(* Logix 5000 project; controller TBEN_Lx_8IOL_AOI_V0_2 vendor 1 type 14 code 176 rev 32.11; software revision 32.00; part 6 of 11 *)

           TBEN_L4_8IOL:C.Data[144].6   // IO-Link Port 8 - Device ID (INT bit22)
           TBEN_L4_8IOL:C.Data[144].7   // IO-Link Port 8 - Device ID (INT bit23)
           TBEN_L4_8IOL:C.Data[145]   // IO-Link Port 8 - Device ID
           TBEN_L4_8IOL:C.Data[145].0   // IO-Link Port 8 - Device ID (INT bit24)
           TBEN_L4_8IOL:C.Data[145].1   // IO-Link Port 8 - Device ID (INT bit25)
           TBEN_L4_8IOL:C.Data[145].2   // IO-Link Port 8 - Device ID (INT bit26)
           TBEN_L4_8IOL:C.Data[145].3   // IO-Link Port 8 - Device ID (INT bit27)
           TBEN_L4_8IOL:C.Data[145].4   // IO-Link Port 8 - Device ID (INT bit28)
           TBEN_L4_8IOL:C.Data[145].5   // IO-Link Port 8 - Device ID (INT bit29)
           TBEN_L4_8IOL:C.Data[145].6   // IO-Link Port 8 - Device ID (INT bit30)
           TBEN_L4_8IOL:C.Data[145].7   // IO-Link Port 8 - Device ID (INT bit31)
           TBEN_L4_8IOL:C.Data[146]   // VAUX1 Pin1 C0 (Ch0/1)
           TBEN_L4_8IOL:C.Data[146].0   // VAUX1 Pin1 C0 (Ch0/1) (ENUM bit0): 00=24 VDC, 01=switchable
           TBEN_L4_8IOL:C.Data[146].1   // VAUX1 Pin1 C0 (Ch0/1) (ENUM bit1): 10=off
           TBEN_L4_8IOL:C.Data[146].2   // Reserved
           TBEN_L4_8IOL:C.Data[146].3   // Reserved
           TBEN_L4_8IOL:C.Data[146].4   // Reserved
           TBEN_L4_8IOL:C.Data[146].5   // Reserved
           TBEN_L4_8IOL:C.Data[146].6   // Reserved
           TBEN_L4_8IOL:C.Data[146].7   // Reserved
           TBEN_L4_8IOL:C.Data[147]   // VAUX1 Pin1 C1 (Ch2/3)
           TBEN_L4_8IOL:C.Data[147].0   // VAUX1 Pin1 C1 (Ch2/3) (ENUM bit0): 00=24 VDC, 01=switchable
           TBEN_L4_8IOL:C.Data[147].1   // VAUX1 Pin1 C1 (Ch2/3) (ENUM bit1): 10=off
           TBEN_L4_8IOL:C.Data[147].2   // Reserved
           TBEN_L4_8IOL:C.Data[147].3   // Reserved
           TBEN_L4_8IOL:C.Data[147].4   // Reserved
           TBEN_L4_8IOL:C.Data[147].5   // Reserved
           TBEN_L4_8IOL:C.Data[147].6   // Reserved
           TBEN_L4_8IOL:C.Data[147].7   // Reserved
           TBEN_L4_8IOL:C.Data[148]   // VAUX1 Pin1 C2 (Ch4/5)
           TBEN_L4_8IOL:C.Data[148].0   // VAUX1 Pin1 C2 (Ch4/5) (ENUM bit0): 00=24 VDC, 01=switchable
           TBEN_L4_8IOL:C.Data[148].1   // VAUX1 Pin1 C2 (Ch4/5) (ENUM bit1): 10=off
           TBEN_L4_8IOL:C.Data[148].2   // Reserved
           TBEN_L4_8IOL:C.Data[148].3   // Reserved
           TBEN_L4_8IOL:C.Data[148].4   // Reserved
           TBEN_L4_8IOL:C.Data[148].5   // Reserved
           TBEN_L4_8IOL:C.Data[148].6   // Reserved
           TBEN_L4_8IOL:C.Data[148].7   // Reserved
           TBEN_L4_8IOL:C.Data[149]   // VAUX1 Pin1 C3 (Ch6/7)
           TBEN_L4_8IOL:C.Data[149].0   // VAUX1 Pin1 C3 (Ch6/7) (ENUM bit0): 00=24 VDC, 01=switchable
           TBEN_L4_8IOL:C.Data[149].1   // VAUX1 Pin1 C3 (Ch6/7) (ENUM bit1): 10=off
           TBEN_L4_8IOL:C.Data[149].2   // Reserved
           TBEN_L4_8IOL:C.Data[149].3   // Reserved
           TBEN_L4_8IOL:C.Data[149].4   // Reserved
           TBEN_L4_8IOL:C.Data[149].5   // Reserved
           TBEN_L4_8IOL:C.Data[149].6   // Reserved
           TBEN_L4_8IOL:C.Data[149].7   // Reserved
           TBEN_L4_8IOL:C.Data[14]   // DXP 1 - Activate output
           TBEN_L4_8IOL:C.Data[14].0   // DXP 1 - Activate output (ENUM bit0): 0=no, 1=yes
           TBEN_L4_8IOL:C.Data[14].1   // Reserved
           TBEN_L4_8IOL:C.Data[14].2   // Reserved
           TBEN_L4_8IOL:C.Data[14].3   // Reserved
           TBEN_L4_8IOL:C.Data[14].4   // Reserved
           TBEN_L4_8IOL:C.Data[14].5   // Reserved
           TBEN_L4_8IOL:C.Data[14].6   // Reserved
           TBEN_L4_8IOL:C.Data[14].7   // Reserved
           TBEN_L4_8IOL:C.Data[150]   // VAUX1 Pin1 C4 (Ch8)
           TBEN_L4_8IOL:C.Data[150].0   // VAUX1 Pin1 C4 (Ch8) (ENUM bit0): 00=24 VDC, 01=switchable
           TBEN_L4_8IOL:C.Data[150].1   // VAUX1 Pin1 C4 (Ch8) (ENUM bit1): 10=off
           TBEN_L4_8IOL:C.Data[150].2   // Reserved
           TBEN_L4_8IOL:C.Data[150].3   // Reserved
           TBEN_L4_8IOL:C.Data[150].4   // Reserved
           TBEN_L4_8IOL:C.Data[150].5   // Reserved
           TBEN_L4_8IOL:C.Data[150].6   // Reserved
           TBEN_L4_8IOL:C.Data[150].7   // Reserved
           TBEN_L4_8IOL:C.Data[151]   // VAUX2 Pin2 C4 (Ch9)
           TBEN_L4_8IOL:C.Data[151].0   // VAUX2 Pin2 C4 (Ch9) (ENUM bit0): 00=24 VDC, 01=switchable
           TBEN_L4_8IOL:C.Data[151].1   // VAUX2 Pin2 C4 (Ch9) (ENUM bit1): 10=off
           TBEN_L4_8IOL:C.Data[151].2   // Reserved
           TBEN_L4_8IOL:C.Data[151].3   // Reserved
           TBEN_L4_8IOL:C.Data[151].4   // Reserved
           TBEN_L4_8IOL:C.Data[151].5   // Reserved
           TBEN_L4_8IOL:C.Data[151].6   // Reserved
           TBEN_L4_8IOL:C.Data[151].7   // Reserved
           TBEN_L4_8IOL:C.Data[152]   // VAUX1 Pin1 C5 (Ch10)
           TBEN_L4_8IOL:C.Data[152].0   // VAUX1 Pin1 C5 (Ch10) (ENUM bit0): 00=24 VDC, 01=switchable
           TBEN_L4_8IOL:C.Data[152].1   // VAUX1 Pin1 C5 (Ch10) (ENUM bit1): 10=off
           TBEN_L4_8IOL:C.Data[152].2   // Reserved
           TBEN_L4_8IOL:C.Data[152].3   // Reserved
           TBEN_L4_8IOL:C.Data[152].4   // Reserved
           TBEN_L4_8IOL:C.Data[152].5   // Reserved
           TBEN_L4_8IOL:C.Data[152].6   // Reserved
           TBEN_L4_8IOL:C.Data[152].7   // Reserved
           TBEN_L4_8IOL:C.Data[153]   // VAUX2 Pin2 C5 (Ch11)
           TBEN_L4_8IOL:C.Data[153].0   // VAUX2 Pin2 C5 (Ch11) (ENUM bit0): 00=24 VDC, 01=switchable
           TBEN_L4_8IOL:C.Data[153].1   // VAUX2 Pin2 C5 (Ch11) (ENUM bit1): 10=off
           TBEN_L4_8IOL:C.Data[153].2   // Reserved
           TBEN_L4_8IOL:C.Data[153].3   // Reserved
           TBEN_L4_8IOL:C.Data[153].4   // Reserved
           TBEN_L4_8IOL:C.Data[153].5   // Reserved
           TBEN_L4_8IOL:C.Data[153].6   // Reserved
           TBEN_L4_8IOL:C.Data[153].7   // Reserved
           TBEN_L4_8IOL:C.Data[154]   // VAUX1 Pin1 C6 (Ch12)
           TBEN_L4_8IOL:C.Data[154].0   // VAUX1 Pin1 C6 (Ch12) (ENUM bit0): 00=24 VDC, 01=switchable
           TBEN_L4_8IOL:C.Data[154].1   // VAUX1 Pin1 C6 (Ch12) (ENUM bit1): 10=off
           TBEN_L4_8IOL:C.Data[154].2   // Reserved
           TBEN_L4_8IOL:C.Data[154].3   // Reserved
           TBEN_L4_8IOL:C.Data[154].4   // Reserved
           TBEN_L4_8IOL:C.Data[154].5   // Reserved
           TBEN_L4_8IOL:C.Data[154].6   // Reserved
           TBEN_L4_8IOL:C.Data[154].7   // Reserved
           TBEN_L4_8IOL:C.Data[155]   // VAUX2 Pin2 C6 (Ch13)
           TBEN_L4_8IOL:C.Data[155].0   // VAUX2 Pin2 C6 (Ch13) (ENUM bit0): 00=24 VDC, 01=switchable
           TBEN_L4_8IOL:C.Data[155].1   // VAUX2 Pin2 C6 (Ch13) (ENUM bit1): 10=off
           TBEN_L4_8IOL:C.Data[155].2   // Reserved
           TBEN_L4_8IOL:C.Data[155].3   // Reserved
           TBEN_L4_8IOL:C.Data[155].4   // Reserved
           TBEN_L4_8IOL:C.Data[155].5   // Reserved
           TBEN_L4_8IOL:C.Data[155].6   // Reserved
           TBEN_L4_8IOL:C.Data[155].7   // Reserved
           TBEN_L4_8IOL:C.Data[156]   // VAUX1 Pin1 C7 (Ch14)
           TBEN_L4_8IOL:C.Data[156].0   // VAUX1 Pin1 C7 (Ch14) (ENUM bit0): 00=24 VDC, 01=switchable
           TBEN_L4_8IOL:C.Data[156].1   // VAUX1 Pin1 C7 (Ch14) (ENUM bit1): 10=off
           TBEN_L4_8IOL:C.Data[156].2   // Reserved
           TBEN_L4_8IOL:C.Data[156].3   // Reserved
           TBEN_L4_8IOL:C.Data[156].4   // Reserved
           TBEN_L4_8IOL:C.Data[156].5   // Reserved
           TBEN_L4_8IOL:C.Data[156].6   // Reserved
           TBEN_L4_8IOL:C.Data[156].7   // Reserved
           TBEN_L4_8IOL:C.Data[157]   // VAUX2 Pin2 C7 (Ch15)
           TBEN_L4_8IOL:C.Data[157].0   // VAUX2 Pin2 C7 (Ch15) (ENUM bit0): 00=24 VDC, 01=switchable
           TBEN_L4_8IOL:C.Data[157].1   // VAUX2 Pin2 C7 (Ch15) (ENUM bit1): 10=off
           TBEN_L4_8IOL:C.Data[157].2   // Reserved
           TBEN_L4_8IOL:C.Data[157].3   // Reserved
           TBEN_L4_8IOL:C.Data[157].4   // Reserved
           TBEN_L4_8IOL:C.Data[157].5   // Reserved
           TBEN_L4_8IOL:C.Data[157].6   // Reserved
           TBEN_L4_8IOL:C.Data[157].7   // Reserved
           TBEN_L4_8IOL:C.Data[15]   // DXP 3 - Activate output
           TBEN_L4_8IOL:C.Data[15].0   // DXP 3 - Activate output (ENUM bit0): 0=no, 1=yes
           TBEN_L4_8IOL:C.Data[15].1   // Reserved
           TBEN_L4_8IOL:C.Data[15].2   // Reserved
           TBEN_L4_8IOL:C.Data[15].3   // Reserved
           TBEN_L4_8IOL:C.Data[15].4   // Reserved
           TBEN_L4_8IOL:C.Data[15].5   // Reserved
           TBEN_L4_8IOL:C.Data[15].6   // Reserved
           TBEN_L4_8IOL:C.Data[15].7   // Reserved
           TBEN_L4_8IOL:C.Data[16]   // DXP 5 - Activate output
           TBEN_L4_8IOL:C.Data[16].0   // DXP 5 - Activate output (ENUM bit0): 0=no, 1=yes
           TBEN_L4_8IOL:C.Data[16].1   // Reserved
           TBEN_L4_8IOL:C.Data[16].2   // Reserved
           TBEN_L4_8IOL:C.Data[16].3   // Reserved
           TBEN_L4_8IOL:C.Data[16].4   // Reserved
           TBEN_L4_8IOL:C.Data[16].5   // Reserved
           TBEN_L4_8IOL:C.Data[16].6   // Reserved
           TBEN_L4_8IOL:C.Data[16].7   // Reserved
           TBEN_L4_8IOL:C.Data[17]   // DXP 7 - Activate output
           TBEN_L4_8IOL:C.Data[17].0   // DXP 7 - Activate output (ENUM bit0): 0=no, 1=yes
           TBEN_L4_8IOL:C.Data[17].1   // Reserved
           TBEN_L4_8IOL:C.Data[17].2   // Reserved
           TBEN_L4_8IOL:C.Data[17].3   // Reserved
           TBEN_L4_8IOL:C.Data[17].4   // Reserved
           TBEN_L4_8IOL:C.Data[17].5   // Reserved
           TBEN_L4_8IOL:C.Data[17].6   // Reserved
           TBEN_L4_8IOL:C.Data[17].7   // Reserved
           TBEN_L4_8IOL:C.Data[18]   // IO-Link Port 1 - Operation mode
           TBEN_L4_8IOL:C.Data[18].0   // IO-Link Port 1 - Operation mode (ENUM bit0): 0000=IO-Link without validation, 0001=IO-Link with family compatible device
           TBEN_L4_8IOL:C.Data[18].1   // IO-Link Port 1 - Operation mode (ENUM bit1): 0010=IO-Link with compatible device, 0011=IO-Link with identical device
           TBEN_L4_8IOL:C.Data[18].2   // IO-Link Port 1 - Operation mode (ENUM bit2): 0100=DI (with parameter access)
           TBEN_L4_8IOL:C.Data[18].3   // IO-Link Port 1 - Operation mode (ENUM bit3): 1000=DI
           TBEN_L4_8IOL:C.Data[18].4   // Reserved
           TBEN_L4_8IOL:C.Data[18].5   // Reserved
           TBEN_L4_8IOL:C.Data[18].6   // Reserved
           TBEN_L4_8IOL:C.Data[18].7   // Reserved
           TBEN_L4_8IOL:C.Data[19]   // IO-Link Port 1 - Data storage mode
           TBEN_L4_8IOL:C.Data[19].0   // IO-Link Port 1 - Data storage mode (ENUM bit0): 00=activated, 01=overwrite
           TBEN_L4_8IOL:C.Data[19].1   // IO-Link Port 1 - Data storage mode (ENUM bit1): 10=read in, 11=deactivated, clear
           TBEN_L4_8IOL:C.Data[19].2   // Reserved
           TBEN_L4_8IOL:C.Data[19].3   // Reserved
           TBEN_L4_8IOL:C.Data[19].4   // Reserved
           TBEN_L4_8IOL:C.Data[19].5   // Reserved
           TBEN_L4_8IOL:C.Data[19].6   // Reserved
           TBEN_L4_8IOL:C.Data[19].7   // Reserved
           TBEN_L4_8IOL:C.Data[1]   // Reserved
           TBEN_L4_8IOL:C.Data[20]   // IO-Link Port 1 - Cycle time
           TBEN_L4_8IOL:C.Data[20].0   // IO-Link Port 1 - Cycle time (ENUM bit0): 00000000=automatic, 00010000=1.6 ms, 00011000=2.4 ms, 00100000=3.2 ms, 00101000=4.0 ms, 00110000=4.8 ms, 00111000=5.6 ms, 01000000=6.4 ms, 01000010=7.2 ms, 01000100=8.0 ms, 01000110=8.8 ms, 01001000=9.6 ms
           TBEN_L4_8IOL:C.Data[20].1   // IO-Link Port 1 - Cycle time (ENUM bit1): 01001010=10.4 ms, 01001100=11.2 ms, 01001110=12.0 ms, 01010000=12.8 ms, 01010100=14.4 ms, 01011000=16.0 ms, 01011100=17.6 ms, 01100000=19.2 ms, 01100100=20.8 ms, 01101000=22.4 ms, 01101100=24.0 ms, 01110000=25.6 ms
           TBEN_L4_8IOL:C.Data[20].2   // IO-Link Port 1 - Cycle time (ENUM bit2): 01110100=27.2 ms, 01111000=28.8 ms, 01111100=30.4 ms, 10000000=32.0 ms, 10000001=33.6 ms, 10000010=35.2 ms, 10000011=36.8 ms, 10000100=38.4 ms, 10000101=40.0 ms, 10000110=41.6 ms, 10000111=43.2 ms, 10001000=44.8 ms
           TBEN_L4_8IOL:C.Data[20].3   // IO-Link Port 1 - Cycle time (ENUM bit3): 10001001=46.4 ms, 10001010=48.0 ms, 10001011=49.6 ms, 10001100=51.2 ms, 10001101=52.8 ms, 10001110=54.4 ms, 10001111=56.0 ms, 10010000=57.6 ms, 10010001=59.2 ms, 10010010=60.8 ms, 10010011=62.4 ms, 10010100=64.0 ms
           TBEN_L4_8IOL:C.Data[20].4   // IO-Link Port 1 - Cycle time (ENUM bit4): 10010101=65.6 ms, 10010110=67.2 ms, 10010111=68.8 ms, 10011000=70.4 ms, 10011001=72.0 ms, 10011010=73.6 ms, 10011011=75.2 ms, 10011100=76.8 ms, 10011101=78.4 ms, 10011110=80.0 ms, 10011111=81.6 ms
           TBEN_L4_8IOL:C.Data[20].5   // IO-Link Port 1 - Cycle time (ENUM bit5): 10100000=83.2 ms, 10100001=84.8 ms, 10100010=86.4 ms, 10100011=88.0 ms, 10100100=89.6 ms, 10100101=91.2 ms, 10100110=92.8 ms, 10100111=94.4 ms, 10101000=96.0 ms, 10101001=97.6 ms, 10101010=99.2 ms
           TBEN_L4_8IOL:C.Data[20].6   // IO-Link Port 1 - Cycle time (ENUM bit6): 10101011=100.8 ms, 10101100=102.4 ms, 10101101=104.0 ms, 10101110=105.6 ms, 10101111=107.2 ms, 10110000=108.8 ms, 10110001=110.4 ms, 10110010=112.0 ms, 10110011=113.6 ms, 10110100=115.2 ms, 10110101=116.8 ms
           TBEN_L4_8IOL:C.Data[20].7   // IO-Link Port 1 - Cycle time (ENUM bit7): 10110110=118.4 ms, 10110111=120.0 ms, 10111000=121.6 ms, 10111001=123.2 ms, 10111010=124.8 ms, 10111011=126.4 ms, 10111100=128.0 ms, 10111101=129.6 ms, 10111110=131.2 ms, 10111111=132.8 ms, 11111111=automatic, compatible
           TBEN_L4_8IOL:C.Data[21]   // IO-Link Port 1 - Revision
           TBEN_L4_8IOL:C.Data[21].0   // IO-Link Port 1 - Revision (ENUM bit0): 0=automatic, 1=V1.0
           TBEN_L4_8IOL:C.Data[21].1   // Reserved
           TBEN_L4_8IOL:C.Data[21].2   // Reserved
           TBEN_L4_8IOL:C.Data[21].3   // Reserved
           TBEN_L4_8IOL:C.Data[21].4   // Reserved
           TBEN_L4_8IOL:C.Data[21].5   // Reserved
           TBEN_L4_8IOL:C.Data[21].6   // Reserved
           TBEN_L4_8IOL:C.Data[21].7   // Reserved
           TBEN_L4_8IOL:C.Data[22]   // IO-Link Port 1 - Activate Quick Start-Up
           TBEN_L4_8IOL:C.Data[22].0   // IO-Link Port 1 - Activate Quick Start-Up (ENUM bit0): 0=no, 1=yes
           TBEN_L4_8IOL:C.Data[22].1   // Reserved
           TBEN_L4_8IOL:C.Data[22].2   // Reserved
           TBEN_L4_8IOL:C.Data[22].3   // Reserved
           TBEN_L4_8IOL:C.Data[22].4   // Reserved
           TBEN_L4_8IOL:C.Data[22].5   // Reserved
           TBEN_L4_8IOL:C.Data[22].6   // Reserved
           TBEN_L4_8IOL:C.Data[22].7   // Reserved
           TBEN_L4_8IOL:C.Data[23]   // IO-Link Port 1 - Device parametrization via GSD
           TBEN_L4_8IOL:C.Data[23].0   // IO-Link Port 1 - Device parametrization via GSD (ENUM bit0): 0=inactive, 1=active
           TBEN_L4_8IOL:C.Data[23].1   // Reserved
           TBEN_L4_8IOL:C.Data[23].2   // Reserved
           TBEN_L4_8IOL:C.Data[23].3   // Reserved
           TBEN_L4_8IOL:C.Data[23].4   // Reserved
           TBEN_L4_8IOL:C.Data[23].5   // Reserved
           TBEN_L4_8IOL:C.Data[23].6   // Reserved
           TBEN_L4_8IOL:C.Data[23].7   // Reserved
           TBEN_L4_8IOL:C.Data[24]   // IO-Link Port 1 - Process input data invalid
           TBEN_L4_8IOL:C.Data[24].0   // IO-Link Port 1 - Process input data invalid (ENUM bit0): 0=diagnostic generated, 1=no diagnostic generated
           TBEN_L4_8IOL:C.Data[24].1   // Reserved
           TBEN_L4_8IOL:C.Data[24].2   // Reserved
           TBEN_L4_8IOL:C.Data[24].3   // Reserved
           TBEN_L4_8IOL:C.Data[24].4   // Reserved
           TBEN_L4_8IOL:C.Data[24].5   // Reserved
           TBEN_L4_8IOL:C.Data[24].6   // Reserved
           TBEN_L4_8IOL:C.Data[24].7   // Reserved
           TBEN_L4_8IOL:C.Data[25]   // IO-Link Port 1 - Deactivate diagnostics
           TBEN_L4_8IOL:C.Data[25].0   // IO-Link Port 1 - Deactivate diagnostics (ENUM bit0): 00=no, 01=notifications
           TBEN_L4_8IOL:C.Data[25].1   // IO-Link Port 1 - Deactivate diagnostics (ENUM bit1): 10=notifications and warnings, 11=yes
           TBEN_L4_8IOL:C.Data[25].2   // Reserved
           TBEN_L4_8IOL:C.Data[25].3   // Reserved
           TBEN_L4_8IOL:C.Data[25].4   // Reserved
           TBEN_L4_8IOL:C.Data[25].5   // Reserved
           TBEN_L4_8IOL:C.Data[25].6   // Reserved
           TBEN_L4_8IOL:C.Data[25].7   // Reserved
           TBEN_L4_8IOL:C.Data[26]   // IO-Link Port 1 - Input data mapping
           TBEN_L4_8IOL:C.Data[26].0   // IO-Link Port 1 - Input data mapping (ENUM bit0): 00=direct, 01=swap 16 bit
           TBEN_L4_8IOL:C.Data[26].1   // IO-Link Port 1 - Input data mapping (ENUM bit1): 10=swap 32 bit, 11=swap
           TBEN_L4_8IOL:C.Data[26].2   // Reserved
           TBEN_L4_8IOL:C.Data[26].3   // Reserved
           TBEN_L4_8IOL:C.Data[26].4   // Reserved
           TBEN_L4_8IOL:C.Data[26].5   // Reserved
           TBEN_L4_8IOL:C.Data[26].6   // Reserved
           TBEN_L4_8IOL:C.Data[26].7   // Reserved
           TBEN_L4_8IOL:C.Data[27]   // IO-Link Port 1 - Output data mapping
           TBEN_L4_8IOL:C.Data[27].0   // IO-Link Port 1 - Output data mapping (ENUM bit0): 00=direct, 01=swap 16 bit
           TBEN_L4_8IOL:C.Data[27].1   // IO-Link Port 1 - Output data mapping (ENUM bit1): 10=swap 32 bit, 11=swap
           TBEN_L4_8IOL:C.Data[27].2   // Reserved
           TBEN_L4_8IOL:C.Data[27].3   // Reserved
           TBEN_L4_8IOL:C.Data[27].4   // Reserved
           TBEN_L4_8IOL:C.Data[27].5   // Reserved
           TBEN_L4_8IOL:C.Data[27].6   // Reserved
           TBEN_L4_8IOL:C.Data[27].7   // Reserved
           TBEN_L4_8IOL:C.Data[28]   // IO-Link Port 1 - Vendor ID
           TBEN_L4_8IOL:C.Data[28].0   // IO-Link Port 1 - Vendor ID (INT bit0)
           TBEN_L4_8IOL:C.Data[28].1   // IO-Link Port 1 - Vendor ID (INT bit1)
           TBEN_L4_8IOL:C.Data[28].2   // IO-Link Port 1 - Vendor ID (INT bit2)
           TBEN_L4_8IOL:C.Data[28].3   // IO-Link Port 1 - Vendor ID (INT bit3)
           TBEN_L4_8IOL:C.Data[28].4   // IO-Link Port 1 - Vendor ID (INT bit4)
           TBEN_L4_8IOL:C.Data[28].5   // IO-Link Port 1 - Vendor ID (INT bit5)
           TBEN_L4_8IOL:C.Data[28].6   // IO-Link Port 1 - Vendor ID (INT bit6)
           TBEN_L4_8IOL:C.Data[28].7   // IO-Link Port 1 - Vendor ID (INT bit7)
           TBEN_L4_8IOL:C.Data[29]   // IO-Link Port 1 - Vendor ID
           TBEN_L4_8IOL:C.Data[29].0   // IO-Link Port 1 - Vendor ID (INT bit8)
           TBEN_L4_8IOL:C.Data[29].1   // IO-Link Port 1 - Vendor ID (INT bit9)
           TBEN_L4_8IOL:C.Data[29].2   // IO-Link Port 1 - Vendor ID (INT bit10)
           TBEN_L4_8IOL:C.Data[29].3   // IO-Link Port 1 - Vendor ID (INT bit11)
           TBEN_L4_8IOL:C.Data[29].4   // IO-Link Port 1 - Vendor ID (INT bit12)
           TBEN_L4_8IOL:C.Data[29].5   // IO-Link Port 1 - Vendor ID (INT bit13)
           TBEN_L4_8IOL:C.Data[29].6   // IO-Link Port 1 - Vendor ID (INT bit14)
           TBEN_L4_8IOL:C.Data[29].7   // IO-Link Port 1 - Vendor ID (INT bit15)
           TBEN_L4_8IOL:C.Data[2]   // Reserved
           TBEN_L4_8IOL:C.Data[30]   // IO-Link Port 1 - Device ID
           TBEN_L4_8IOL:C.Data[30].0   // IO-Link Port 1 - Device ID (INT bit0)
           TBEN_L4_8IOL:C.Data[30].1   // IO-Link Port 1 - Device ID (INT bit1)
           TBEN_L4_8IOL:C.Data[30].2   // IO-Link Port 1 - Device ID (INT bit2)
           TBEN_L4_8IOL:C.Data[30].3   // IO-Link Port 1 - Device ID (INT bit3)
           TBEN_L4_8IOL:C.Data[30].4   // IO-Link Port 1 - Device ID (INT bit4)
           TBEN_L4_8IOL:C.Data[30].5   // IO-Link Port 1 - Device ID (INT bit5)
           TBEN_L4_8IOL:C.Data[30].6   // IO-Link Port 1 - Device ID (INT bit6)
           TBEN_L4_8IOL:C.Data[30].7   // IO-Link Port 1 - Device ID (INT bit7)
           TBEN_L4_8IOL:C.Data[31]   // IO-Link Port 1 - Device ID
           TBEN_L4_8IOL:C.Data[31].0   // IO-Link Port 1 - Device ID (INT bit8)
           TBEN_L4_8IOL:C.Data[31].1   // IO-Link Port 1 - Device ID (INT bit9)
           TBEN_L4_8IOL:C.Data[31].2   // IO-Link Port 1 - Device ID (INT bit10)
           TBEN_L4_8IOL:C.Data[31].3   // IO-Link Port 1 - Device ID (INT bit11)
           TBEN_L4_8IOL:C.Data[31].4   // IO-Link Port 1 - Device ID (INT bit12)
           TBEN_L4_8IOL:C.Data[31].5   // IO-Link Port 1 - Device ID (INT bit13)
           TBEN_L4_8IOL:C.Data[31].6   // IO-Link Port 1 - Device ID (INT bit14)
           TBEN_L4_8IOL:C.Data[31].7   // IO-Link Port 1 - Device ID (INT bit15)
           TBEN_L4_8IOL:C.Data[32]   // IO-Link Port 1 - Device ID
           TBEN_L4_8IOL:C.Data[32].0   // IO-Link Port 1 - Device ID (INT bit16)
           TBEN_L4_8IOL:C.Data[32].1   // IO-Link Port 1 - Device ID (INT bit17)
           TBEN_L4_8IOL:C.Data[32].2   // IO-Link Port 1 - Device ID (INT bit18)
           TBEN_L4_8IOL:C.Data[32].3   // IO-Link Port 1 - Device ID (INT bit19)
           TBEN_L4_8IOL:C.Data[32].4   // IO-Link Port 1 - Device ID (INT bit20)
           TBEN_L4_8IOL:C.Data[32].5   // IO-Link Port 1 - Device ID (INT bit21)
           TBEN_L4_8IOL:C.Data[32].6   // IO-Link Port 1 - Device ID (INT bit22)
           TBEN_L4_8IOL:C.Data[32].7   // IO-Link Port 1 - Device ID (INT bit23)
           TBEN_L4_8IOL:C.Data[33]   // IO-Link Port 1 - Device ID
           TBEN_L4_8IOL:C.Data[33].0   // IO-Link Port 1 - Device ID (INT bit24)
           TBEN_L4_8IOL:C.Data[33].1   // IO-Link Port 1 - Device ID (INT bit25)
           TBEN_L4_8IOL:C.Data[33].2   // IO-Link Port 1 - Device ID (INT bit26)
           TBEN_L4_8IOL:C.Data[33].3   // IO-Link Port 1 - Device ID (INT bit27)
           TBEN_L4_8IOL:C.Data[33].4   // IO-Link Port 1 - Device ID (INT bit28)
           TBEN_L4_8IOL:C.Data[33].5   // IO-Link Port 1 - Device ID (INT bit29)
           TBEN_L4_8IOL:C.Data[33].6   // IO-Link Port 1 - Device ID (INT bit30)
           TBEN_L4_8IOL:C.Data[33].7   // IO-Link Port 1 - Device ID (INT bit31)
           TBEN_L4_8IOL:C.Data[34]   // IO-Link Port 2 - Operation mode
           TBEN_L4_8IOL:C.Data[34].0   // IO-Link Port 2 - Operation mode (ENUM bit0): 0000=IO-Link without validation, 0001=IO-Link with family compatible device
           TBEN_L4_8IOL:C.Data[34].1   // IO-Link Port 2 - Operation mode (ENUM bit1): 0010=IO-Link with compatible device, 0011=IO-Link with identical device
           TBEN_L4_8IOL:C.Data[34].2   // IO-Link Port 2 - Operation mode (ENUM bit2): 0100=DI (with parameter access)
           TBEN_L4_8IOL:C.Data[34].3   // IO-Link Port 2 - Operation mode (ENUM bit3): 1000=DI
           TBEN_L4_8IOL:C.Data[34].4   // Reserved
           TBEN_L4_8IOL:C.Data[34].5   // Reserved
           TBEN_L4_8IOL:C.Data[34].6   // Reserved
           TBEN_L4_8IOL:C.Data[34].7   // Reserved
           TBEN_L4_8IOL:C.Data[35]   // IO-Link Port 2 - Data storage mode
           TBEN_L4_8IOL:C.Data[35].0   // IO-Link Port 2 - Data storage mode (ENUM bit0): 00=activated, 01=overwrite
           TBEN_L4_8IOL:C.Data[35].1   // IO-Link Port 2 - Data storage mode (ENUM bit1): 10=read in, 11=deactivated, clear
           TBEN_L4_8IOL:C.Data[35].2   // Reserved
           TBEN_L4_8IOL:C.Data[35].3   // Reserved
           TBEN_L4_8IOL:C.Data[35].4   // Reserved
           TBEN_L4_8IOL:C.Data[35].5   // Reserved
           TBEN_L4_8IOL:C.Data[35].6   // Reserved
           TBEN_L4_8IOL:C.Data[35].7   // Reserved
           TBEN_L4_8IOL:C.Data[36]   // IO-Link Port 2 - Cycle time
           TBEN_L4_8IOL:C.Data[36].0   // IO-Link Port 2 - Cycle time (ENUM bit0): 00000000=automatic, 00010000=1.6 ms, 00011000=2.4 ms, 00100000=3.2 ms, 00101000=4.0 ms, 00110000=4.8 ms, 00111000=5.6 ms, 01000000=6.4 ms, 01000010=7.2 ms, 01000100=8.0 ms, 01000110=8.8 ms, 01001000=9.6 ms
           TBEN_L4_8IOL:C.Data[36].1   // IO-Link Port 2 - Cycle time (ENUM bit1): 01001010=10.4 ms, 01001100=11.2 ms, 01001110=12.0 ms, 01010000=12.8 ms, 01010100=14.4 ms, 01011000=16.0 ms, 01011100=17.6 ms, 01100000=19.2 ms, 01100100=20.8 ms, 01101000=22.4 ms, 01101100=24.0 ms, 01110000=25.6 ms
           TBEN_L4_8IOL:C.Data[36].2   // IO-Link Port 2 - Cycle time (ENUM bit2): 01110100=27.2 ms, 01111000=28.8 ms, 01111100=30.4 ms, 10000000=32.0 ms, 10000001=33.6 ms, 10000010=35.2 ms, 10000011=36.8 ms, 10000100=38.4 ms, 10000101=40.0 ms, 10000110=41.6 ms, 10000111=43.2 ms, 10001000=44.8 ms
           TBEN_L4_8IOL:C.Data[36].3   // IO-Link Port 2 - Cycle time (ENUM bit3): 10001001=46.4 ms, 10001010=48.0 ms, 10001011=49.6 ms, 10001100=51.2 ms, 10001101=52.8 ms, 10001110=54.4 ms, 10001111=56.0 ms, 10010000=57.6 ms, 10010001=59.2 ms, 10010010=60.8 ms, 10010011=62.4 ms, 10010100=64.0 ms
           TBEN_L4_8IOL:C.Data[36].4   // IO-Link Port 2 - Cycle time (ENUM bit4): 10010101=65.6 ms, 10010110=67.2 ms, 10010111=68.8 ms, 10011000=70.4 ms, 10011001=72.0 ms, 10011010=73.6 ms, 10011011=75.2 ms, 10011100=76.8 ms, 10011101=78.4 ms, 10011110=80.0 ms, 10011111=81.6 ms
           TBEN_L4_8IOL:C.Data[36].5   // IO-Link Port 2 - Cycle time (ENUM bit5): 10100000=83.2 ms, 10100001=84.8 ms, 10100010=86.4 ms, 10100011=88.0 ms, 10100100=89.6 ms, 10100101=91.2 ms, 10100110=92.8 ms, 10100111=94.4 ms, 10101000=96.0 ms, 10101001=97.6 ms, 10101010=99.2 ms
           TBEN_L4_8IOL:C.Data[36].6   // IO-Link Port 2 - Cycle time (ENUM bit6): 10101011=100.8 ms, 10101100=102.4 ms, 10101101=104.0 ms, 10101110=105.6 ms, 10101111=107.2 ms, 10110000=108.8 ms, 10110001=110.4 ms, 10110010=112.0 ms, 10110011=113.6 ms, 10110100=115.2 ms, 10110101=116.8 ms
           TBEN_L4_8IOL:C.Data[36].7   // IO-Link Port 2 - Cycle time (ENUM bit7): 10110110=118.4 ms, 10110111=120.0 ms, 10111000=121.6 ms, 10111001=123.2 ms, 10111010=124.8 ms, 10111011=126.4 ms, 10111100=128.0 ms, 10111101=129.6 ms, 10111110=131.2 ms, 10111111=132.8 ms, 11111111=automatic, compatible
           TBEN_L4_8IOL:C.Data[37]   // IO-Link Port 2 - Revision
           TBEN_L4_8IOL:C.Data[37].0   // IO-Link Port 2 - Revision (ENUM bit0): 0=automatic, 1=V1.0
           TBEN_L4_8IOL:C.Data[37].1   // Reserved
           TBEN_L4_8IOL:C.Data[37].2   // Reserved
           TBEN_L4_8IOL:C.Data[37].3   // Reserved
           TBEN_L4_8IOL:C.Data[37].4   // Reserved
           TBEN_L4_8IOL:C.Data[37].5   // Reserved
           TBEN_L4_8IOL:C.Data[37].6   // Reserved
           TBEN_L4_8IOL:C.Data[37].7   // Reserved
           TBEN_L4_8IOL:C.Data[38]   // IO-Link Port 2 - Activate Quick Start-Up
           TBEN_L4_8IOL:C.Data[38].0   // IO-Link Port 2 - Activate Quick Start-Up (ENUM bit0): 0=no, 1=yes
           TBEN_L4_8IOL:C.Data[38].1   // Reserved
           TBEN_L4_8IOL:C.Data[38].2   // Reserved
           TBEN_L4_8IOL:C.Data[38].3   // Reserved
           TBEN_L4_8IOL:C.Data[38].4   // Reserved
           TBEN_L4_8IOL:C.Data[38].5   // Reserved
           TBEN_L4_8IOL:C.Data[38].6   // Reserved
           TBEN_L4_8IOL:C.Data[38].7   // Reserved
           TBEN_L4_8IOL:C.Data[39]   // IO-Link Port 2 - Device parametrization via GSD
           TBEN_L4_8IOL:C.Data[39].0   // IO-Link Port 2 - Device parametrization via GSD (ENUM bit0): 0=inactive, 1=active
           TBEN_L4_8IOL:C.Data[39].1   // Reserved
           TBEN_L4_8IOL:C.Data[39].2   // Reserved
           TBEN_L4_8IOL:C.Data[39].3   // Reserved
           TBEN_L4_8IOL:C.Data[39].4   // Reserved
           TBEN_L4_8IOL:C.Data[39].5   // Reserved
           TBEN_L4_8IOL:C.Data[39].6   // Reserved
           TBEN_L4_8IOL:C.Data[39].7   // Reserved
           TBEN_L4_8IOL:C.Data[3]   // Reserved
           TBEN_L4_8IOL:C.Data[40]   // IO-Link Port 2 - Process input data invalid
           TBEN_L4_8IOL:C.Data[40].0   // IO-Link Port 2 - Process input data invalid (ENUM bit0): 0=diagnostic generated, 1=no diagnostic generated
           TBEN_L4_8IOL:C.Data[40].1   // Reserved
           TBEN_L4_8IOL:C.Data[40].2   // Reserved
           TBEN_L4_8IOL:C.Data[40].3   // Reserved
           TBEN_L4_8IOL:C.Data[40].4   // Reserved
           TBEN_L4_8IOL:C.Data[40].5   // Reserved
           TBEN_L4_8IOL:C.Data[40].6   // Reserved
           TBEN_L4_8IOL:C.Data[40].7   // Reserved
           TBEN_L4_8IOL:C.Data[41]   // IO-Link Port 2 - Deactivate diagnostics
           TBEN_L4_8IOL:C.Data[41].0   // IO-Link Port 2 - Deactivate diagnostics (ENUM bit0): 00=no, 01=notifications
           TBEN_L4_8IOL:C.Data[41].1   // IO-Link Port 2 - Deactivate diagnostics (ENUM bit1): 10=notifications and warnings, 11=yes
           TBEN_L4_8IOL:C.Data[41].2   // Reserved
           TBEN_L4_8IOL:C.Data[41].3   // Reserved
           TBEN_L4_8IOL:C.Data[41].4   // Reserved
           TBEN_L4_8IOL:C.Data[41].5   // Reserved
           TBEN_L4_8IOL:C.Data[41].6   // Reserved
           TBEN_L4_8IOL:C.Data[41].7   // Reserved
           TBEN_L4_8IOL:C.Data[42]   // IO-Link Port 2 - Input data mapping
           TBEN_L4_8IOL:C.Data[42].0   // IO-Link Port 2 - Input data mapping (ENUM bit0): 00=direct, 01=swap 16 bit
           TBEN_L4_8IOL:C.Data[42].1   // IO-Link Port 2 - Input data mapping (ENUM bit1): 10=swap 32 bit, 11=swap
           TBEN_L4_8IOL:C.Data[42].2   // Reserved
           TBEN_L4_8IOL:C.Data[42].3   // Reserved
           TBEN_L4_8IOL:C.Data[42].4   // Reserved
           TBEN_L4_8IOL:C.Data[42].5   // Reserved
           TBEN_L4_8IOL:C.Data[42].6   // Reserved
           TBEN_L4_8IOL:C.Data[42].7   // Reserved
           TBEN_L4_8IOL:C.Data[43]   // IO-Link Port 2 - Output data mapping
           TBEN_L4_8IOL:C.Data[43].0   // IO-Link Port 2 - Output data mapping (ENUM bit0): 00=direct, 01=swap 16 bit
           TBEN_L4_8IOL:C.Data[43].1   // IO-Link Port 2 - Output data mapping (ENUM bit1): 10=swap 32 bit, 11=swap
           TBEN_L4_8IOL:C.Data[43].2   // Reserved
           TBEN_L4_8IOL:C.Data[43].3   // Reserved
           TBEN_L4_8IOL:C.Data[43].4   // Reserved
           TBEN_L4_8IOL:C.Data[43].5   // Reserved
           TBEN_L4_8IOL:C.Data[43].6   // Reserved
           TBEN_L4_8IOL:C.Data[43].7   // Reserved
           TBEN_L4_8IOL:C.Data[44]   // IO-Link Port 2 - Vendor ID
           TBEN_L4_8IOL:C.Data[44].0   // IO-Link Port 2 - Vendor ID (INT bit0)
           TBEN_L4_8IOL:C.Data[44].1   // IO-Link Port 2 - Vendor ID (INT bit1)
           TBEN_L4_8IOL:C.Data[44].2   // IO-Link Port 2 - Vendor ID (INT bit2)
           TBEN_L4_8IOL:C.Data[44].3   // IO-Link Port 2 - Vendor ID (INT bit3)
           TBEN_L4_8IOL:C.Data[44].4   // IO-Link Port 2 - Vendor ID (INT bit4)
           TBEN_L4_8IOL:C.Data[44].5   // IO-Link Port 2 - Vendor ID (INT bit5)
           TBEN_L4_8IOL:C.Data[44].6   // IO-Link Port 2 - Vendor ID (INT bit6)
           TBEN_L4_8IOL:C.Data[44].7   // IO-Link Port 2 - Vendor ID (INT bit7)
           TBEN_L4_8IOL:C.Data[45]   // IO-Link Port 2 - Vendor ID
           TBEN_L4_8IOL:C.Data[45].0   // IO-Link Port 2 - Vendor ID (INT bit8)
           TBEN_L4_8IOL:C.Data[45].1   // IO-Link Port 2 - Vendor ID (INT bit9)
           TBEN_L4_8IOL:C.Data[45].2   // IO-Link Port 2 - Vendor ID (INT bit10)
           TBEN_L4_8IOL:C.Data[45].3   // IO-Link Port 2 - Vendor ID (INT bit11)
           TBEN_L4_8IOL:C.Data[45].4   // IO-Link Port 2 - Vendor ID (INT bit12)
           TBEN_L4_8IOL:C.Data[45].5   // IO-Link Port 2 - Vendor ID (INT bit13)
           TBEN_L4_8IOL:C.Data[45].6   // IO-Link Port 2 - Vendor ID (INT bit14)
           TBEN_L4_8IOL:C.Data[45].7   // IO-Link Port 2 - Vendor ID (INT bit15)
           TBEN_L4_8IOL:C.Data[46]   // IO-Link Port 2 - Device ID
           TBEN_L4_8IOL:C.Data[46].0   // IO-Link Port 2 - Device ID (INT bit0)
           TBEN_L4_8IOL:C.Data[46].1   // IO-Link Port 2 - Device ID (INT bit1)
           TBEN_L4_8IOL:C.Data[46].2   // IO-Link Port 2 - Device ID (INT bit2)
           TBEN_L4_8IOL:C.Data[46].3   // IO-Link Port 2 - Device ID (INT bit3)
           TBEN_L4_8IOL:C.Data[46].4   // IO-Link Port 2 - Device ID (INT bit4)
           TBEN_L4_8IOL:C.Data[46].5   // IO-Link Port 2 - Device ID (INT bit5)
           TBEN_L4_8IOL:C.Data[46].6   // IO-Link Port 2 - Device ID (INT bit6)
           TBEN_L4_8IOL:C.Data[46].7   // IO-Link Port 2 - Device ID (INT bit7)
           TBEN_L4_8IOL:C.Data[47]   // IO-Link Port 2 - Device ID
           TBEN_L4_8IOL:C.Data[47].0   // IO-Link Port 2 - Device ID (INT bit8)
           TBEN_L4_8IOL:C.Data[47].1   // IO-Link Port 2 - Device ID (INT bit9)
           TBEN_L4_8IOL:C.Data[47].2   // IO-Link Port 2 - Device ID (INT bit10)
           TBEN_L4_8IOL:C.Data[47].3   // IO-Link Port 2 - Device ID (INT bit11)
           TBEN_L4_8IOL:C.Data[47].4   // IO-Link Port 2 - Device ID (INT bit12)
           TBEN_L4_8IOL:C.Data[47].5   // IO-Link Port 2 - Device ID (INT bit13)
           TBEN_L4_8IOL:C.Data[47].6   // IO-Link Port 2 - Device ID (INT bit14)
           TBEN_L4_8IOL:C.Data[47].7   // IO-Link Port 2 - Device ID (INT bit15)
           TBEN_L4_8IOL:C.Data[48]   // IO-Link Port 2 - Device ID
           TBEN_L4_8IOL:C.Data[48].0   // IO-Link Port 2 - Device ID (INT bit16)
           TBEN_L4_8IOL:C.Data[48].1   // IO-Link Port 2 - Device ID (INT bit17)
           TBEN_L4_8IOL:C.Data[48].2   // IO-Link Port 2 - Device ID (INT bit18)
           TBEN_L4_8IOL:C.Data[48].3   // IO-Link Port 2 - Device ID (INT bit19)
           TBEN_L4_8IOL:C.Data[48].4   // IO-Link Port 2 - Device ID (INT bit20)
           TBEN_L4_8IOL:C.Data[48].5   // IO-Link Port 2 - Device ID (INT bit21)
           TBEN_L4_8IOL:C.Data[48].6   // IO-Link Port 2 - Device ID (INT bit22)
           TBEN_L4_8IOL:C.Data[48].7   // IO-Link Port 2 - Device ID (INT bit23)
           TBEN_L4_8IOL:C.Data[49]   // IO-Link Port 2 - Device ID
           TBEN_L4_8IOL:C.Data[49].0   // IO-Link Port 2 - Device ID (INT bit24)
           TBEN_L4_8IOL:C.Data[49].1   // IO-Link Port 2 - Device ID (INT bit25)
           TBEN_L4_8IOL:C.Data[49].2   // IO-Link Port 2 - Device ID (INT bit26)
           TBEN_L4_8IOL:C.Data[49].3   // IO-Link Port 2 - Device ID (INT bit27)
           TBEN_L4_8IOL:C.Data[49].4   // IO-Link Port 2 - Device ID (INT bit28)
           TBEN_L4_8IOL:C.Data[49].5   // IO-Link Port 2 - Device ID (INT bit29)
           TBEN_L4_8IOL:C.Data[49].6   // IO-Link Port 2 - Device ID (INT bit30)
           TBEN_L4_8IOL:C.Data[49].7   // IO-Link Port 2 - Device ID (INT bit31)
           TBEN_L4_8IOL:C.Data[4]   // Reserved
           TBEN_L4_8IOL:C.Data[50]   // IO-Link Port 3 - Operation mode
           TBEN_L4_8IOL:C.Data[50].0   // IO-Link Port 3 - Operation mode (ENUM bit0): 0000=IO-Link without validation, 0001=IO-Link with family compatible device
           TBEN_L4_8IOL:C.Data[50].1   // IO-Link Port 3 - Operation mode (ENUM bit1): 0010=IO-Link with compatible device, 0011=IO-Link with identical device
           TBEN_L4_8IOL:C.Data[50].2   // IO-Link Port 3 - Operation mode (ENUM bit2): 0100=DI (with parameter access)
           TBEN_L4_8IOL:C.Data[50].3   // IO-Link Port 3 - Operation mode (ENUM bit3): 1000=DI
           TBEN_L4_8IOL:C.Data[50].4   // Reserved
           TBEN_L4_8IOL:C.Data[50].5   // Reserved
           TBEN_L4_8IOL:C.Data[50].6   // Reserved
           TBEN_L4_8IOL:C.Data[50].7   // Reserved
           TBEN_L4_8IOL:C.Data[51]   // IO-Link Port 3 - Data storage mode
           TBEN_L4_8IOL:C.Data[51].0   // IO-Link Port 3 - Data storage mode (ENUM bit0): 00=activated, 01=overwrite
           TBEN_L4_8IOL:C.Data[51].1   // IO-Link Port 3 - Data storage mode (ENUM bit1): 10=read in, 11=deactivated, clear
           TBEN_L4_8IOL:C.Data[51].2   // Reserved
           TBEN_L4_8IOL:C.Data[51].3   // Reserved
           TBEN_L4_8IOL:C.Data[51].4   // Reserved
           TBEN_L4_8IOL:C.Data[51].5   // Reserved
           TBEN_L4_8IOL:C.Data[51].6   // Reserved
           TBEN_L4_8IOL:C.Data[51].7   // Reserved
           TBEN_L4_8IOL:C.Data[52]   // IO-Link Port 3 - Cycle time
           TBEN_L4_8IOL:C.Data[52].0   // IO-Link Port 3 - Cycle time (ENUM bit0): 00000000=automatic, 00010000=1.6 ms, 00011000=2.4 ms, 00100000=3.2 ms, 00101000=4.0 ms, 00110000=4.8 ms, 00111000=5.6 ms, 01000000=6.4 ms, 01000010=7.2 ms, 01000100=8.0 ms, 01000110=8.8 ms, 01001000=9.6 ms
           TBEN_L4_8IOL:C.Data[52].1   // IO-Link Port 3 - Cycle time (ENUM bit1): 01001010=10.4 ms, 01001100=11.2 ms, 01001110=12.0 ms, 01010000=12.8 ms, 01010100=14.4 ms, 01011000=16.0 ms, 01011100=17.6 ms, 01100000=19.2 ms, 01100100=20.8 ms, 01101000=22.4 ms, 01101100=24.0 ms, 01110000=25.6 ms
           TBEN_L4_8IOL:C.Data[52].2   // IO-Link Port 3 - Cycle time (ENUM bit2): 01110100=27.2 ms, 01111000=28.8 ms, 01111100=30.4 ms, 10000000=32.0 ms, 10000001=33.6 ms, 10000010=35.2 ms, 10000011=36.8 ms, 10000100=38.4 ms, 10000101=40.0 ms, 10000110=41.6 ms, 10000111=43.2 ms, 10001000=44.8 ms
           TBEN_L4_8IOL:C.Data[52].3   // IO-Link Port 3 - Cycle time (ENUM bit3): 10001001=46.4 ms, 10001010=48.0 ms, 10001011=49.6 ms, 10001100=51.2 ms, 10001101=52.8 ms, 10001110=54.4 ms, 10001111=56.0 ms, 10010000=57.6 ms, 10010001=59.2 ms, 10010010=60.8 ms, 10010011=62.4 ms, 10010100=64.0 ms
           TBEN_L4_8IOL:C.Data[52].4   // IO-Link Port 3 - Cycle time (ENUM bit4): 10010101=65.6 ms, 10010110=67.2 ms, 10010111=68.8 ms, 10011000=70.4 ms, 10011001=72.0 ms, 10011010=73.6 ms, 10011011=75.2 ms, 10011100=76.8 ms, 10011101=78.4 ms, 10011110=80.0 ms, 10011111=81.6 ms
           TBEN_L4_8IOL:C.Data[52].5   // IO-Link Port 3 - Cycle time (ENUM bit5): 10100000=83.2 ms, 10100001=84.8 ms, 10100010=86.4 ms, 10100011=88.0 ms, 10100100=89.6 ms, 10100101=91.2 ms, 10100110=92.8 ms, 10100111=94.4 ms, 10101000=96.0 ms, 10101001=97.6 ms, 10101010=99.2 ms
           TBEN_L4_8IOL:C.Data[52].6   // IO-Link Port 3 - Cycle time (ENUM bit6): 10101011=100.8 ms, 10101100=102.4 ms, 10101101=104.0 ms, 10101110=105.6 ms, 10101111=107.2 ms, 10110000=108.8 ms, 10110001=110.4 ms, 10110010=112.0 ms, 10110011=113.6 ms, 10110100=115.2 ms, 10110101=116.8 ms
           TBEN_L4_8IOL:C.Data[52].7   // IO-Link Port 3 - Cycle time (ENUM bit7): 10110110=118.4 ms, 10110111=120.0 ms, 10111000=121.6 ms, 10111001=123.2 ms, 10111010=124.8 ms, 10111011=126.4 ms, 10111100=128.0 ms, 10111101=129.6 ms, 10111110=131.2 ms, 10111111=132.8 ms, 11111111=automatic, compatible
           TBEN_L4_8IOL:C.Data[53]   // IO-Link Port 3 - Revision
           TBEN_L4_8IOL:C.Data[53].0   // IO-Link Port 3 - Revision (ENUM bit0): 0=automatic, 1=V1.0
           TBEN_L4_8IOL:C.Data[53].1   // Reserved
           TBEN_L4_8IOL:C.Data[53].2   // Reserved
           TBEN_L4_8IOL:C.Data[53].3   // Reserved
           TBEN_L4_8IOL:C.Data[53].4   // Reserved
           TBEN_L4_8IOL:C.Data[53].5   // Reserved
           TBEN_L4_8IOL:C.Data[53].6   // Reserved
           TBEN_L4_8IOL:C.Data[53].7   // Reserved
           TBEN_L4_8IOL:C.Data[54]   // IO-Link Port 3 - Activate Quick Start-Up
           TBEN_L4_8IOL:C.Data[54].0   // IO-Link Port 3 - Activate Quick Start-Up (ENUM bit0): 0=no, 1=yes
           TBEN_L4_8IOL:C.Data[54].1   // Reserved
           TBEN_L4_8IOL:C.Data[54].2   // Reserved
           TBEN_L4_8IOL:C.Data[54].3   // Reserved
           TBEN_L4_8IOL:C.Data[54].4   // Reserved
           TBEN_L4_8IOL:C.Data[54].5   // Reserved
           TBEN_L4_8IOL:C.Data[54].6   // Reserved
           TBEN_L4_8IOL:C.Data[54].7   // Reserved
           TBEN_L4_8IOL:C.Data[55]   // IO-Link Port 3 - Device parametrization via GSD
           TBEN_L4_8IOL:C.Data[55].0   // IO-Link Port 3 - Device parametrization via GSD (ENUM bit0): 0=inactive, 1=active
           TBEN_L4_8IOL:C.Data[55].1   // Reserved
           TBEN_L4_8IOL:C.Data[55].2   // Reserved
           TBEN_L4_8IOL:C.Data[55].3   // Reserved
           TBEN_L4_8IOL:C.Data[55].4   // Reserved
           TBEN_L4_8IOL:C.Data[55].5   // Reserved
           TBEN_L4_8IOL:C.Data[55].6   // Reserved
           TBEN_L4_8IOL:C.Data[55].7   // Reserved
           TBEN_L4_8IOL:C.Data[56]   // IO-Link Port 3 - Process input data invalid
           TBEN_L4_8IOL:C.Data[56].0   // IO-Link Port 3 - Process input data invalid (ENUM bit0): 0=diagnostic generated, 1=no diagnostic generated
           TBEN_L4_8IOL:C.Data[56].1   // Reserved
           TBEN_L4_8IOL:C.Data[56].2   // Reserved
           TBEN_L4_8IOL:C.Data[56].3   // Reserved
           TBEN_L4_8IOL:C.Data[56].4   // Reserved
           TBEN_L4_8IOL:C.Data[56].5   // Reserved
           TBEN_L4_8IOL:C.Data[56].6   // Reserved
           TBEN_L4_8IOL:C.Data[56].7   // Reserved
           TBEN_L4_8IOL:C.Data[57]   // IO-Link Port 3 - Deactivate diagnostics
           TBEN_L4_8IOL:C.Data[57].0   // IO-Link Port 3 - Deactivate diagnostics (ENUM bit0): 00=no, 01=notifications
           TBEN_L4_8IOL:C.Data[57].1   // IO-Link Port 3 - Deactivate diagnostics (ENUM bit1): 10=notifications and warnings, 11=yes
           TBEN_L4_8IOL:C.Data[57].2   // Reserved
           TBEN_L4_8IOL:C.Data[57].3   // Reserved
           TBEN_L4_8IOL:C.Data[57].4   // Reserved
           TBEN_L4_8IOL:C.Data[57].5   // Reserved
           TBEN_L4_8IOL:C.Data[57].6   // Reserved
           TBEN_L4_8IOL:C.Data[57].7   // Reserved
           TBEN_L4_8IOL:C.Data[58]   // IO-Link Port 3 - Input data mapping
           TBEN_L4_8IOL:C.Data[58].0   // IO-Link Port 3 - Input data mapping (ENUM bit0): 00=direct, 01=swap 16 bit
           TBEN_L4_8IOL:C.Data[58].1   // IO-Link Port 3 - Input data mapping (ENUM bit1): 10=swap 32 bit, 11=swap
           TBEN_L4_8IOL:C.Data[58].2   // Reserved
           TBEN_L4_8IOL:C.Data[58].3   // Reserved
           TBEN_L4_8IOL:C.Data[58].4   // Reserved
           TBEN_L4_8IOL:C.Data[58].5   // Reserved
           TBEN_L4_8IOL:C.Data[58].6   // Reserved
           TBEN_L4_8IOL:C.Data[58].7   // Reserved
           TBEN_L4_8IOL:C.Data[59]   // IO-Link Port 3 - Output data mapping
           TBEN_L4_8IOL:C.Data[59].0   // IO-Link Port 3 - Output data mapping (ENUM bit0): 00=direct, 01=swap 16 bit
           TBEN_L4_8IOL:C.Data[59].1   // IO-Link Port 3 - Output data mapping (ENUM bit1): 10=swap 32 bit, 11=swap
           TBEN_L4_8IOL:C.Data[59].2   // Reserved
           TBEN_L4_8IOL:C.Data[59].3   // Reserved
           TBEN_L4_8IOL:C.Data[59].4   // Reserved
           TBEN_L4_8IOL:C.Data[59].5   // Reserved
           TBEN_L4_8IOL:C.Data[59].6   // Reserved
           TBEN_L4_8IOL:C.Data[59].7   // Reserved
           TBEN_L4_8IOL:C.Data[5]   // Reserved
           TBEN_L4_8IOL:C.Data[60]   // IO-Link Port 3 - Vendor ID
           TBEN_L4_8IOL:C.Data[60].0   // IO-Link Port 3 - Vendor ID (INT bit0)
           TBEN_L4_8IOL:C.Data[60].1   // IO-Link Port 3 - Vendor ID (INT bit1)
           TBEN_L4_8IOL:C.Data[60].2   // IO-Link Port 3 - Vendor ID (INT bit2)
           TBEN_L4_8IOL:C.Data[60].3   // IO-Link Port 3 - Vendor ID (INT bit3)
           TBEN_L4_8IOL:C.Data[60].4   // IO-Link Port 3 - Vendor ID (INT bit4)
           TBEN_L4_8IOL:C.Data[60].5   // IO-Link Port 3 - Vendor ID (INT bit5)
           TBEN_L4_8IOL:C.Data[60].6   // IO-Link Port 3 - Vendor ID (INT bit6)
           TBEN_L4_8IOL:C.Data[60].7   // IO-Link Port 3 - Vendor ID (INT bit7)
           TBEN_L4_8IOL:C.Data[61]   // IO-Link Port 3 - Vendor ID
           TBEN_L4_8IOL:C.Data[61].0   // IO-Link Port 3 - Vendor ID (INT bit8)
           TBEN_L4_8IOL:C.Data[61].1   // IO-Link Port 3 - Vendor ID (INT bit9)
           TBEN_L4_8IOL:C.Data[61].2   // IO-Link Port 3 - Vendor ID (INT bit10)
           TBEN_L4_8IOL:C.Data[61].3   // IO-Link Port 3 - Vendor ID (INT bit11)
           TBEN_L4_8IOL:C.Data[61].4   // IO-Link Port 3 - Vendor ID (INT bit12)
           TBEN_L4_8IOL:C.Data[61].5   // IO-Link Port 3 - Vendor ID (INT bit13)
           TBEN_L4_8IOL:C.Data[61].6   // IO-Link Port 3 - Vendor ID (INT bit14)
           TBEN_L4_8IOL:C.Data[61].7   // IO-Link Port 3 - Vendor ID (INT bit15)
           TBEN_L4_8IOL:C.Data[62]   // IO-Link Port 3 - Device ID
           TBEN_L4_8IOL:C.Data[62].0   // IO-Link Port 3 - Device ID (INT bit0)
           TBEN_L4_8IOL:C.Data[62].1   // IO-Link Port 3 - Device ID (INT bit1)
           TBEN_L4_8IOL:C.Data[62].2   // IO-Link Port 3 - Device ID (INT bit2)
           TBEN_L4_8IOL:C.Data[62].3   // IO-Link Port 3 - Device ID (INT bit3)
           TBEN_L4_8IOL:C.Data[62].4   // IO-Link Port 3 - Device ID (INT bit4)
           TBEN_L4_8IOL:C.Data[62].5   // IO-Link Port 3 - Device ID (INT bit5)
           TBEN_L4_8IOL:C.Data[62].6   // IO-Link Port 3 - Device ID (INT bit6)
           TBEN_L4_8IOL:C.Data[62].7   // IO-Link Port 3 - Device ID (INT bit7)
           TBEN_L4_8IOL:C.Data[63]   // IO-Link Port 3 - Device ID
           TBEN_L4_8IOL:C.Data[63].0   // IO-Link Port 3 - Device ID (INT bit8)
           TBEN_L4_8IOL:C.Data[63].1   // IO-Link Port 3 - Device ID (INT bit9)
           TBEN_L4_8IOL:C.Data[63].2   // IO-Link Port 3 - Device ID (INT bit10)
           TBEN_L4_8IOL:C.Data[63].3   // IO-Link Port 3 - Device ID (INT bit11)
           TBEN_L4_8IOL:C.Data[63].4   // IO-Link Port 3 - Device ID (INT bit12)
           TBEN_L4_8IOL:C.Data[63].5   // IO-Link Port 3 - Device ID (INT bit13)
           TBEN_L4_8IOL:C.Data[63].6   // IO-Link Port 3 - Device ID (INT bit14)
           TBEN_L4_8IOL:C.Data[63].7   // IO-Link Port 3 - Device ID (INT bit15)
           TBEN_L4_8IOL:C.Data[64]   // IO-Link Port 3 - Device ID
           TBEN_L4_8IOL:C.Data[64].0   // IO-Link Port 3 - Device ID (INT bit16)
           TBEN_L4_8IOL:C.Data[64].1   // IO-Link Port 3 - Device ID (INT bit17)
           TBEN_L4_8IOL:C.Data[64].2   // IO-Link Port 3 - Device ID (INT bit18)
           TBEN_L4_8IOL:C.Data[64].3   // IO-Link Port 3 - Device ID (INT bit19)
           TBEN_L4_8IOL:C.Data[64].4   // IO-Link Port 3 - Device ID (INT bit20)
           TBEN_L4_8IOL:C.Data[64].5   // IO-Link Port 3 - Device ID (INT bit21)
           TBEN_L4_8IOL:C.Data[64].6   // IO-Link Port 3 - Device ID (INT bit22)
           TBEN_L4_8IOL:C.Data[64].7   // IO-Link Port 3 - Device ID (INT bit23)
           TBEN_L4_8IOL:C.Data[65]   // IO-Link Port 3 - Device ID
           TBEN_L4_8IOL:C.Data[65].0   // IO-Link Port 3 - Device ID (INT bit24)
           TBEN_L4_8IOL:C.Data[65].1   // IO-Link Port 3 - Device ID (INT bit25)
           TBEN_L4_8IOL:C.Data[65].2   // IO-Link Port 3 - Device ID (INT bit26)
           TBEN_L4_8IOL:C.Data[65].3   // IO-Link Port 3 - Device ID (INT bit27)
           TBEN_L4_8IOL:C.Data[65].4   // IO-Link Port 3 - Device ID (INT bit28)
           TBEN_L4_8IOL:C.Data[65].5   // IO-Link Port 3 - Device ID (INT bit29)
           TBEN_L4_8IOL:C.Data[65].6   // IO-Link Port 3 - Device ID (INT bit30)
           TBEN_L4_8IOL:C.Data[65].7   // IO-Link Port 3 - Device ID (INT bit31)
           TBEN_L4_8IOL:C.Data[66]   // IO-Link Port 4 - Operation mode
           TBEN_L4_8IOL:C.Data[66].0   // IO-Link Port 4 - Operation mode (ENUM bit0): 0000=IO-Link without validation, 0001=IO-Link with family compatible device
           TBEN_L4_8IOL:C.Data[66].1   // IO-Link Port 4 - Operation mode (ENUM bit1): 0010=IO-Link with compatible device, 0011=IO-Link with identical device
           TBEN_L4_8IOL:C.Data[66].2   // IO-Link Port 4 - Operation mode (ENUM bit2): 0100=DI (with parameter access)
           TBEN_L4_8IOL:C.Data[66].3   // IO-Link Port 4 - Operation mode (ENUM bit3): 1000=DI
           TBEN_L4_8IOL:C.Data[66].4   // Reserved
           TBEN_L4_8IOL:C.Data[66].5   // Reserved
           TBEN_L4_8IOL:C.Data[66].6   // Reserved
           TBEN_L4_8IOL:C.Data[66].7   // Reserved
           TBEN_L4_8IOL:C.Data[67]   // IO-Link Port 4 - Data storage mode
           TBEN_L4_8IOL:C.Data[67].0   // IO-Link Port 4 - Data storage mode (ENUM bit0): 00=activated, 01=overwrite
           TBEN_L4_8IOL:C.Data[67].1   // IO-Link Port 4 - Data storage mode (ENUM bit1): 10=read in, 11=deactivated, clear
           TBEN_L4_8IOL:C.Data[67].2   // Reserved
           TBEN_L4_8IOL:C.Data[67].3   // Reserved
           TBEN_L4_8IOL:C.Data[67].4   // Reserved
           TBEN_L4_8IOL:C.Data[67].5   // Reserved
           TBEN_L4_8IOL:C.Data[67].6   // Reserved
           TBEN_L4_8IOL:C.Data[67].7   // Reserved
           TBEN_L4_8IOL:C.Data[68]   // IO-Link Port 4 - Cycle time
           TBEN_L4_8IOL:C.Data[68].0   // IO-Link Port 4 - Cycle time (ENUM bit0): 00000000=automatic, 00010000=1.6 ms, 00011000=2.4 ms, 00100000=3.2 ms, 00101000=4.0 ms, 00110000=4.8 ms, 00111000=5.6 ms, 01000000=6.4 ms, 01000010=7.2 ms, 01000100=8.0 ms, 01000110=8.8 ms, 01001000=9.6 ms
           TBEN_L4_8IOL:C.Data[68].1   // IO-Link Port 4 - Cycle time (ENUM bit1): 01001010=10.4 ms, 01001100=11.2 ms, 01001110=12.0 ms, 01010000=12.8 ms, 01010100=14.4 ms, 01011000=16.0 ms, 01011100=17.6 ms, 01100000=19.2 ms, 01100100=20.8 ms, 01101000=22.4 ms, 01101100=24.0 ms, 01110000=25.6 ms
           TBEN_L4_8IOL:C.Data[68].2   // IO-Link Port 4 - Cycle time (ENUM bit2): 01110100=27.2 ms, 01111000=28.8 ms, 01111100=30.4 ms, 10000000=32.0 ms, 10000001=33.6 ms, 10000010=35.2 ms, 10000011=36.8 ms, 10000100=38.4 ms, 10000101=40.0 ms, 10000110=41.6 ms, 10000111=43.2 ms, 10001000=44.8 ms
           TBEN_L4_8IOL:C.Data[68].3   // IO-Link Port 4 - Cycle time (ENUM bit3): 10001001=46.4 ms, 10001010=48.0 ms, 10001011=49.6 ms, 10001100=51.2 ms, 10001101=52.8 ms, 10001110=54.4 ms, 10001111=56.0 ms, 10010000=57.6 ms, 10010001=59.2 ms, 10010010=60.8 ms, 10010011=62.4 ms, 10010100=64.0 ms
           TBEN_L4_8IOL:C.Data[68].4   // IO-Link Port 4 - Cycle time (ENUM bit4): 10010101=65.6 ms, 10010110=67.2 ms, 10010111=68.8 ms, 10011000=70.4 ms, 10011001=72.0 ms, 10011010=73.6 ms, 10011011=75.2 ms, 10011100=76.8 ms, 10011101=78.4 ms, 10011110=80.0 ms, 10011111=81.6 ms
           TBEN_L4_8IOL:C.Data[68].5   // IO-Link Port 4 - Cycle time (ENUM bit5): 10100000=83.2 ms, 10100001=84.8 ms, 10100010=86.4 ms, 10100011=88.0 ms, 10100100=89.6 ms, 10100101=91.2 ms, 10100110=92.8 ms, 10100111=94.4 ms, 10101000=96.0 ms, 10101001=97.6 ms, 10101010=99.2 ms
           TBEN_L4_8IOL:C.Data[68].6   // IO-Link Port 4 - Cycle time (ENUM bit6): 10101011=100.8 ms, 10101100=102.4 ms, 10101101=104.0 ms, 10101110=105.6 ms, 10101111=107.2 ms, 10110000=108.8 ms, 10110001=110.4 ms, 10110010=112.0 ms, 10110011=113.6 ms, 10110100=115.2 ms, 10110101=116.8 ms
           TBEN_L4_8IOL:C.Data[68].7   // IO-Link Port 4 - Cycle time (ENUM bit7): 10110110=118.4 ms, 10110111=120.0 ms, 10111000=121.6 ms, 10111001=123.2 ms, 10111010=124.8 ms, 10111011=126.4 ms, 10111100=128.0 ms, 10111101=129.6 ms, 10111110=131.2 ms, 10111111=132.8 ms, 11111111=automatic, compatible
           TBEN_L4_8IOL:C.Data[69]   // IO-Link Port 4 - Revision
           TBEN_L4_8IOL:C.Data[69].0   // IO-Link Port 4 - Revision (ENUM bit0): 0=automatic, 1=V1.0
           TBEN_L4_8IOL:C.Data[69].1   // Reserved
           TBEN_L4_8IOL:C.Data[69].2   // Reserved
           TBEN_L4_8IOL:C.Data[69].3   // Reserved
           TBEN_L4_8IOL:C.Data[69].4   // Reserved
           TBEN_L4_8IOL:C.Data[69].5   // Reserved
           TBEN_L4_8IOL:C.Data[69].6   // Reserved
           TBEN_L4_8IOL:C.Data[69].7   // Reserved
           TBEN_L4_8IOL:C.Data[6]   // Reserved
           TBEN_L4_8IOL:C.Data[70]   // IO-Link Port 4 - Activate Quick Start-Up
           TBEN_L4_8IOL:C.Data[70].0   // IO-Link Port 4 - Activate Quick Start-Up (ENUM bit0): 0=no, 1=yes
           TBEN_L4_8IOL:C.Data[70].1   // Reserved
           TBEN_L4_8IOL:C.Data[70].2   // Reserved
           TBEN_L4_8IOL:C.Data[70].3   // Reserved
           TBEN_L4_8IOL:C.Data[70].4   // Reserved
           TBEN_L4_8IOL:C.Data[70].5   // Reserved
           TBEN_L4_8IOL:C.Data[70].6   // Reserved
           TBEN_L4_8IOL:C.Data[70].7   // Reserved
           TBEN_L4_8IOL:C.Data[71]   // IO-Link Port 4 - Device parametrization via GSD
           TBEN_L4_8IOL:C.Data[71].0   // IO-Link Port 4 - Device parametrization via GSD (ENUM bit0): 0=inactive, 1=active
           TBEN_L4_8IOL:C.Data[71].1   // Reserved
           TBEN_L4_8IOL:C.Data[71].2   // Reserved
           TBEN_L4_8IOL:C.Data[71].3   // Reserved
           TBEN_L4_8IOL:C.Data[71].4   // Reserved
           TBEN_L4_8IOL:C.Data[71].5   // Reserved
           TBEN_L4_8IOL:C.Data[71].6   // Reserved
           TBEN_L4_8IOL:C.Data[71].7   // Reserved
           TBEN_L4_8IOL:C.Data[72]   // IO-Link Port 4 - Process input data invalid
           TBEN_L4_8IOL:C.Data[72].0   // IO-Link Port 4 - Process input data invalid (ENUM bit0): 0=diagnostic generated, 1=no diagnostic generated
           TBEN_L4_8IOL:C.Data[72].1   // Reserved
           TBEN_L4_8IOL:C.Data[72].2   // Reserved
           TBEN_L4_8IOL:C.Data[72].3   // Reserved
           TBEN_L4_8IOL:C.Data[72].4   // Reserved
           TBEN_L4_8IOL:C.Data[72].5   // Reserved
           TBEN_L4_8IOL:C.Data[72].6   // Reserved
           TBEN_L4_8IOL:C.Data[72].7   // Reserved
           TBEN_L4_8IOL:C.Data[73]   // IO-Link Port 4 - Deactivate diagnostics
           TBEN_L4_8IOL:C.Data[73].0   // IO-Link Port 4 - Deactivate diagnostics (ENUM bit0): 00=no, 01=notifications
           TBEN_L4_8IOL:C.Data[73].1   // IO-Link Port 4 - Deactivate diagnostics (ENUM bit1): 10=notifications and warnings, 11=yes
           TBEN_L4_8IOL:C.Data[73].2   // Reserved
           TBEN_L4_8IOL:C.Data[73].3   // Reserved
           TBEN_L4_8IOL:C.Data[73].4   // Reserved
           TBEN_L4_8IOL:C.Data[73].5   // Reserved
           TBEN_L4_8IOL:C.Data[73].6   // Reserved
           TBEN_L4_8IOL:C.Data[73].7   // Reserved
           TBEN_L4_8IOL:C.Data[74]   // IO-Link Port 4 - Input data mapping
           TBEN_L4_8IOL:C.Data[74].0   // IO-Link Port 4 - Input data mapping (ENUM bit0): 00=direct, 01=swap 16 bit
           TBEN_L4_8IOL:C.Data[74].1   // IO-Link Port 4 - Input data mapping (ENUM bit1): 10=swap 32 bit, 11=swap
           TBEN_L4_8IOL:C.Data[74].2   // Reserved
           TBEN_L4_8IOL:C.Data[74].3   // Reserved
           TBEN_L4_8IOL:C.Data[74].4   // Reserved
           TBEN_L4_8IOL:C.Data[74].5   // Reserved
           TBEN_L4_8IOL:C.Data[74].6   // Reserved
           TBEN_L4_8IOL:C.Data[74].7   // Reserved
           TBEN_L4_8IOL:C.Data[75]   // IO-Link Port 4 - Output data mapping
           TBEN_L4_8IOL:C.Data[75].0   // IO-Link Port 4 - Output data mapping (ENUM bit0): 00=direct, 01=swap 16 bit
           TBEN_L4_8IOL:C.Data[75].1   // IO-Link Port 4 - Output data mapping (ENUM bit1): 10=swap 32 bit, 11=swap
           TBEN_L4_8IOL:C.Data[75].2   // Reserved
           TBEN_L4_8IOL:C.Data[75].3   // Reserved
           TBEN_L4_8IOL:C.Data[75].4   // Reserved
           TBEN_L4_8IOL:C.Data[75].5   // Reserved
           TBEN_L4_8IOL:C.Data[75].6   // Reserved
           TBEN_L4_8IOL:C.Data[75].7   // Reserved
           TBEN_L4_8IOL:C.Data[76]   // IO-Link Port 4 - Vendor ID
           TBEN_L4_8IOL:C.Data[76].0   // IO-Link Port 4 - Vendor ID (INT bit0)
           TBEN_L4_8IOL:C.Data[76].1   // IO-Link Port 4 - Vendor ID (INT bit1)
           TBEN_L4_8IOL:C.Data[76].2   // IO-Link Port 4 - Vendor ID (INT bit2)
           TBEN_L4_8IOL:C.Data[76].3   // IO-Link Port 4 - Vendor ID (INT bit3)
           TBEN_L4_8IOL:C.Data[76].4   // IO-Link Port 4 - Vendor ID (INT bit4)
           TBEN_L4_8IOL:C.Data[76].5   // IO-Link Port 4 - Vendor ID (INT bit5)
           TBEN_L4_8IOL:C.Data[76].6   // IO-Link Port 4 - Vendor ID (INT bit6)
           TBEN_L4_8IOL:C.Data[76].7   // IO-Link Port 4 - Vendor ID (INT bit7)
           TBEN_L4_8IOL:C.Data[77]   // IO-Link Port 4 - Vendor ID
           TBEN_L4_8IOL:C.Data[77].0   // IO-Link Port 4 - Vendor ID (INT bit8)
           TBEN_L4_8IOL:C.Data[77].1   // IO-Link Port 4 - Vendor ID (INT bit9)
           TBEN_L4_8IOL:C.Data[77].2   // IO-Link Port 4 - Vendor ID (INT bit10)
           TBEN_L4_8IOL:C.Data[77].3   // IO-Link Port 4 - Vendor ID (INT bit11)
           TBEN_L4_8IOL:C.Data[77].4   // IO-Link Port 4 - Vendor ID (INT bit12)
           TBEN_L4_8IOL:C.Data[77].5   // IO-Link Port 4 - Vendor ID (INT bit13)
           TBEN_L4_8IOL:C.Data[77].6   // IO-Link Port 4 - Vendor ID (INT bit14)
           TBEN_L4_8IOL:C.Data[77].7   // IO-Link Port 4 - Vendor ID (INT bit15)
           TBEN_L4_8IOL:C.Data[78]   // IO-Link Port 4 - Device ID
           TBEN_L4_8IOL:C.Data[78].0   // IO-Link Port 4 - Device ID (INT bit0)
           TBEN_L4_8IOL:C.Data[78].1   // IO-Link Port 4 - Device ID (INT bit1)
           TBEN_L4_8IOL:C.Data[78].2   // IO-Link Port 4 - Device ID (INT bit2)
           TBEN_L4_8IOL:C.Data[78].3   // IO-Link Port 4 - Device ID (INT bit3)
           TBEN_L4_8IOL:C.Data[78].4   // IO-Link Port 4 - Device ID (INT bit4)
           TBEN_L4_8IOL:C.Data[78].5   // IO-Link Port 4 - Device ID (INT bit5)
           TBEN_L4_8IOL:C.Data[78].6   // IO-Link Port 4 - Device ID (INT bit6)
           TBEN_L4_8IOL:C.Data[78].7   // IO-Link Port 4 - Device ID (INT bit7)
           TBEN_L4_8IOL:C.Data[79]   // IO-Link Port 4 - Device ID
           TBEN_L4_8IOL:C.Data[79].0   // IO-Link Port 4 - Device ID (INT bit8)
           TBEN_L4_8IOL:C.Data[79].1   // IO-Link Port 4 - Device ID (INT bit9)
           TBEN_L4_8IOL:C.Data[79].2   // IO-Link Port 4 - Device ID (INT bit10)
           TBEN_L4_8IOL:C.Data[79].3   // IO-Link Port 4 - Device ID (INT bit11)
           TBEN_L4_8IOL:C.Data[79].4   // IO-Link Port 4 - Device ID (INT bit12)
           TBEN_L4_8IOL:C.Data[79].5   // IO-Link Port 4 - Device ID (INT bit13)
           TBEN_L4_8IOL:C.Data[79].6   // IO-Link Port 4 - Device ID (INT bit14)
           TBEN_L4_8IOL:C.Data[79].7   // IO-Link Port 4 - Device ID (INT bit15)
           TBEN_L4_8IOL:C.Data[7]   // Reserved
           TBEN_L4_8IOL:C.Data[80]   // IO-Link Port 4 - Device ID
           TBEN_L4_8IOL:C.Data[80].0   // IO-Link Port 4 - Device ID (INT bit16)
           TBEN_L4_8IOL:C.Data[80].1   // IO-Link Port 4 - Device ID (INT bit17)
           TBEN_L4_8IOL:C.Data[80].2   // IO-Link Port 4 - Device ID (INT bit18)
           TBEN_L4_8IOL:C.Data[80].3   // IO-Link Port 4 - Device ID (INT bit19)
           TBEN_L4_8IOL:C.Data[80].4   // IO-Link Port 4 - Device ID (INT bit20)
           TBEN_L4_8IOL:C.Data[80].5   // IO-Link Port 4 - Device ID (INT bit21)
           TBEN_L4_8IOL:C.Data[80].6   // IO-Link Port 4 - Device ID (INT bit22)
           TBEN_L4_8IOL:C.Data[80].7   // IO-Link Port 4 - Device ID (INT bit23)
           TBEN_L4_8IOL:C.Data[81]   // IO-Link Port 4 - Device ID
           TBEN_L4_8IOL:C.Data[81].0   // IO-Link Port 4 - Device ID (INT bit24)
           TBEN_L4_8IOL:C.Data[81].1   // IO-Link Port 4 - Device ID (INT bit25)
           TBEN_L4_8IOL:C.Data[81].2   // IO-Link Port 4 - Device ID (INT bit26)
           TBEN_L4_8IOL:C.Data[81].3   // IO-Link Port 4 - Device ID (INT bit27)
           TBEN_L4_8IOL:C.Data[81].4   // IO-Link Port 4 - Device ID (INT bit28)
           TBEN_L4_8IOL:C.Data[81].5   // IO-Link Port 4 - Device ID (INT bit29)
           TBEN_L4_8IOL:C.Data[81].6   // IO-Link Port 4 - Device ID (INT bit30)
           TBEN_L4_8IOL:C.Data[81].7   // IO-Link Port 4 - Device ID (INT bit31)
           TBEN_L4_8IOL:C.Data[82]   // IO-Link Port 5 - Operation mode
           TBEN_L4_8IOL:C.Data[82].0   // IO-Link Port 5 - Operation mode (ENUM bit0): 0000=IO-Link without validation, 0001=IO-Link with family compatible device
           TBEN_L4_8IOL:C.Data[82].1   // IO-Link Port 5 - Operation mode (ENUM bit1): 0010=IO-Link with compatible device, 0011=IO-Link with identical device
           TBEN_L4_8IOL:C.Data[82].2   // IO-Link Port 5 - Operation mode (ENUM bit2): 0100=DI (with parameter access)
           TBEN_L4_8IOL:C.Data[82].3   // IO-Link Port 5 - Operation mode (ENUM bit3): 1000=DI
           TBEN_L4_8IOL:C.Data[82].4   // Reserved
           TBEN_L4_8IOL:C.Data[82].5   // Reserved
           TBEN_L4_8IOL:C.Data[82].6   // Reserved
           TBEN_L4_8IOL:C.Data[82].7   // Reserved
           TBEN_L4_8IOL:C.Data[83]   // IO-Link Port 5 - Data storage mode
           TBEN_L4_8IOL:C.Data[83].0   // IO-Link Port 5 - Data storage mode (ENUM bit0): 00=activated, 01=overwrite
           TBEN_L4_8IOL:C.Data[83].1   // IO-Link Port 5 - Data storage mode (ENUM bit1): 10=read in, 11=deactivated, clear
           TBEN_L4_8IOL:C.Data[83].2   // Reserved
           TBEN_L4_8IOL:C.Data[83].3   // Reserved
           TBEN_L4_8IOL:C.Data[83].4   // Reserved
           TBEN_L4_8IOL:C.Data[83].5   // Reserved
           TBEN_L4_8IOL:C.Data[83].6   // Reserved
           TBEN_L4_8IOL:C.Data[83].7   // Reserved
           TBEN_L4_8IOL:C.Data[84]   // IO-Link Port 5 - Cycle time
           TBEN_L4_8IOL:C.Data[84].0   // IO-Link Port 5 - Cycle time (ENUM bit0): 00000000=automatic, 00010000=1.6 ms, 00011000=2.4 ms, 00100000=3.2 ms, 00101000=4.0 ms, 00110000=4.8 ms, 00111000=5.6 ms, 01000000=6.4 ms, 01000010=7.2 ms, 01000100=8.0 ms, 01000110=8.8 ms, 01001000=9.6 ms
           TBEN_L4_8IOL:C.Data[84].1   // IO-Link Port 5 - Cycle time (ENUM bit1): 01001010=10.4 ms, 01001100=11.2 ms, 01001110=12.0 ms, 01010000=12.8 ms, 01010100=14.4 ms, 01011000=16.0 ms, 01011100=17.6 ms, 01100000=19.2 ms, 01100100=20.8 ms, 01101000=22.4 ms, 01101100=24.0 ms, 01110000=25.6 ms
           TBEN_L4_8IOL:C.Data[84].2   // IO-Link Port 5 - Cycle time (ENUM bit2): 01110100=27.2 ms, 01111000=28.8 ms, 01111100=30.4 ms, 10000000=32.0 ms, 10000001=33.6 ms, 10000010=35.2 ms, 10000011=36.8 ms, 10000100=38.4 ms, 10000101=40.0 ms, 10000110=41.6 ms, 10000111=43.2 ms, 10001000=44.8 ms
           TBEN_L4_8IOL:C.Data[84].3   // IO-Link Port 5 - Cycle time (ENUM bit3): 10001001=46.4 ms, 10001010=48.0 ms, 10001011=49.6 ms, 10001100=51.2 ms, 10001101=52.8 ms, 10001110=54.4 ms, 10001111=56.0 ms, 10010000=57.6 ms, 10010001=59.2 ms, 10010010=60.8 ms, 10010011=62.4 ms, 10010100=64.0 ms
           TBEN_L4_8IOL:C.Data[84].4   // IO-Link Port 5 - Cycle time (ENUM bit4): 10010101=65.6 ms, 10010110=67.2 ms, 10010111=68.8 ms, 10011000=70.4 ms, 10011001=72.0 ms, 10011010=73.6 ms, 10011011=75.2 ms, 10011100=76.8 ms, 10011101=78.4 ms, 10011110=80.0 ms, 10011111=81.6 ms
           TBEN_L4_8IOL:C.Data[84].5   // IO-Link Port 5 - Cycle time (ENUM bit5): 10100000=83.2 ms, 10100001=84.8 ms, 10100010=86.4 ms, 10100011=88.0 ms, 10100100=89.6 ms, 10100101=91.2 ms, 10100110=92.8 ms, 10100111=94.4 ms, 10101000=96.0 ms, 10101001=97.6 ms, 10101010=99.2 ms
           TBEN_L4_8IOL:C.Data[84].6   // IO-Link Port 5 - Cycle time (ENUM bit6): 10101011=100.8 ms, 10101100=102.4 ms, 10101101=104.0 ms, 10101110=105.6 ms, 10101111=107.2 ms, 10110000=108.8 ms, 10110001=110.4 ms, 10110010=112.0 ms, 10110011=113.6 ms, 10110100=115.2 ms, 10110101=116.8 ms
           TBEN_L4_8IOL:C.Data[84].7   // IO-Link Port 5 - Cycle time (ENUM bit7): 10110110=118.4 ms, 10110111=120.0 ms, 10111000=121.6 ms, 10111001=123.2 ms, 10111010=124.8 ms, 10111011=126.4 ms, 10111100=128.0 ms, 10111101=129.6 ms, 10111110=131.2 ms, 10111111=132.8 ms, 11111111=automatic, compatible
           TBEN_L4_8IOL:C.Data[85]   // IO-Link Port 5 - Revision
           TBEN_L4_8IOL:C.Data[85].0   // IO-Link Port 5 - Revision (ENUM bit0): 0=automatic, 1=V1.0
           TBEN_L4_8IOL:C.Data[85].1   // Reserved
           TBEN_L4_8IOL:C.Data[85].2   // Reserved
           TBEN_L4_8IOL:C.Data[85].3   // Reserved
           TBEN_L4_8IOL:C.Data[85].4   // Reserved
           TBEN_L4_8IOL:C.Data[85].5   // Reserved
           TBEN_L4_8IOL:C.Data[85].6   // Reserved
           TBEN_L4_8IOL:C.Data[85].7   // Reserved
           TBEN_L4_8IOL:C.Data[86]   // IO-Link Port 5 - Activate Quick Start-Up
           TBEN_L4_8IOL:C.Data[86].0   // IO-Link Port 5 - Activate Quick Start-Up (ENUM bit0): 0=no, 1=yes
           TBEN_L4_8IOL:C.Data[86].1   // Reserved
           TBEN_L4_8IOL:C.Data[86].2   // Reserved
           TBEN_L4_8IOL:C.Data[86].3   // Reserved
           TBEN_L4_8IOL:C.Data[86].4   // Reserved
           TBEN_L4_8IOL:C.Data[86].5   // Reserved
           TBEN_L4_8IOL:C.Data[86].6   // Reserved
           TBEN_L4_8IOL:C.Data[86].7   // Reserved
           TBEN_L4_8IOL:C.Data[87]   // IO-Link Port 5 - Device parametrization via GSD
           TBEN_L4_8IOL:C.Data[87].0   // IO-Link Port 5 - Device parametrization via GSD (ENUM bit0): 0=inactive, 1=active
           TBEN_L4_8IOL:C.Data[87].1   // Reserved
           TBEN_L4_8IOL:C.Data[87].2   // Reserved
           TBEN_L4_8IOL:C.Data[87].3   // Reserved
           TBEN_L4_8IOL:C.Data[87].4   // Reserved
           TBEN_L4_8IOL:C.Data[87].5   // Reserved
           TBEN_L4_8IOL:C.Data[87].6   // Reserved
           TBEN_L4_8IOL:C.Data[87].7   // Reserved
           TBEN_L4_8IOL:C.Data[88]   // IO-Link Port 5 - Process input data invalid
           TBEN_L4_8IOL:C.Data[88].0   // IO-Link Port 5 - Process input data invalid (ENUM bit0): 0=diagnostic generated, 1=no diagnostic generated
           TBEN_L4_8IOL:C.Data[88].1   // Reserved
           TBEN_L4_8IOL:C.Data[88].2   // Reserved
           TBEN_L4_8IOL:C.Data[88].3   // Reserved
           TBEN_L4_8IOL:C.Data[88].4   // Reserved
           TBEN_L4_8IOL:C.Data[88].5   // Reserved
           TBEN_L4_8IOL:C.Data[88].6   // Reserved
           TBEN_L4_8IOL:C.Data[88].7   // Reserved
           TBEN_L4_8IOL:C.Data[89]   // IO-Link Port 5 - Deactivate diagnostics
           TBEN_L4_8IOL:C.Data[89].0   // IO-Link Port 5 - Deactivate diagnostics (ENUM bit0): 00=no, 01=notifications
           TBEN_L4_8IOL:C.Data[89].1   // IO-Link Port 5 - Deactivate diagnostics (ENUM bit1): 10=notifications and warnings, 11=yes
           TBEN_L4_8IOL:C.Data[89].2   // Reserved
           TBEN_L4_8IOL:C.Data[89].3   // Reserved
           TBEN_L4_8IOL:C.Data[89].4   // Reserved
           TBEN_L4_8IOL:C.Data[89].5   // Reserved
           TBEN_L4_8IOL:C.Data[89].6   // Reserved
           TBEN_L4_8IOL:C.Data[89].7   // Reserved
           TBEN_L4_8IOL:C.Data[8]   // Reserved
           TBEN_L4_8IOL:C.Data[90]   // IO-Link Port 5 - Input data mapping
           TBEN_L4_8IOL:C.Data[90].0   // IO-Link Port 5 - Input data mapping (ENUM bit0): 00=direct, 01=swap 16 bit
           TBEN_L4_8IOL:C.Data[90].1   // IO-Link Port 5 - Input data mapping (ENUM bit1): 10=swap 32 bit, 11=swap
           TBEN_L4_8IOL:C.Data[90].2   // Reserved
           TBEN_L4_8IOL:C.Data[90].3   // Reserved
           TBEN_L4_8IOL:C.Data[90].4   // Reserved
           TBEN_L4_8IOL:C.Data[90].5   // Reserved
           TBEN_L4_8IOL:C.Data[90].6   // Reserved
           TBEN_L4_8IOL:C.Data[90].7   // Reserved
           TBEN_L4_8IOL:C.Data[91]   // IO-Link Port 5 - Output data mapping
           TBEN_L4_8IOL:C.Data[91].0   // IO-Link Port 5 - Output data mapping (ENUM bit0): 00=direct, 01=swap 16 bit
           TBEN_L4_8IOL:C.Data[91].1   // IO-Link Port 5 - Output data mapping (ENUM bit1): 10=swap 32 bit, 11=swap
           TBEN_L4_8IOL:C.Data[91].2   // Reserved
           TBEN_L4_8IOL:C.Data[91].3   // Reserved
           TBEN_L4_8IOL:C.Data[91].4   // Reserved
           TBEN_L4_8IOL:C.Data[91].5   // Reserved
           TBEN_L4_8IOL:C.Data[91].6   // Reserved
           TBEN_L4_8IOL:C.Data[91].7   // Reserved
           TBEN_L4_8IOL:C.Data[92]   // IO-Link Port 5 - Vendor ID
           TBEN_L4_8IOL:C.Data[92].0   // IO-Link Port 5 - Vendor ID (INT bit0)
           TBEN_L4_8IOL:C.Data[92].1   // IO-Link Port 5 - Vendor ID (INT bit1)
           TBEN_L4_8IOL:C.Data[92].2   // IO-Link Port 5 - Vendor ID (INT bit2)
           TBEN_L4_8IOL:C.Data[92].3   // IO-Link Port 5 - Vendor ID (INT bit3)
           TBEN_L4_8IOL:C.Data[92].4   // IO-Link Port 5 - Vendor ID (INT bit4)
           TBEN_L4_8IOL:C.Data[92].5   // IO-Link Port 5 - Vendor ID (INT bit5)
           TBEN_L4_8IOL:C.Data[92].6   // IO-Link Port 5 - Vendor ID (INT bit6)
           TBEN_L4_8IOL:C.Data[92].7   // IO-Link Port 5 - Vendor ID (INT bit7)
           TBEN_L4_8IOL:C.Data[93]   // IO-Link Port 5 - Vendor ID
           TBEN_L4_8IOL:C.Data[93].0   // IO-Link Port 5 - Vendor ID (INT bit8)
           TBEN_L4_8IOL:C.Data[93].1   // IO-Link Port 5 - Vendor ID (INT bit9)
           TBEN_L4_8IOL:C.Data[93].2   // IO-Link Port 5 - Vendor ID (INT bit10)
           TBEN_L4_8IOL:C.Data[93].3   // IO-Link Port 5 - Vendor ID (INT bit11)
           TBEN_L4_8IOL:C.Data[93].4   // IO-Link Port 5 - Vendor ID (INT bit12)
           TBEN_L4_8IOL:C.Data[93].5   // IO-Link Port 5 - Vendor ID (INT bit13)
           TBEN_L4_8IOL:C.Data[93].6   // IO-Link Port 5 - Vendor ID (INT bit14)
           TBEN_L4_8IOL:C.Data[93].7   // IO-Link Port 5 - Vendor ID (INT bit15)
           TBEN_L4_8IOL:C.Data[94]   // IO-Link Port 5 - Device ID
           TBEN_L4_8IOL:C.Data[94].0   // IO-Link Port 5 - Device ID (INT bit0)
           TBEN_L4_8IOL:C.Data[94].1   // IO-Link Port 5 - Device ID (INT bit1)
           TBEN_L4_8IOL:C.Data[94].2   // IO-Link Port 5 - Device ID (INT bit2)
           TBEN_L4_8IOL:C.Data[94].3   // IO-Link Port 5 - Device ID (INT bit3)
           TBEN_L4_8IOL:C.Data[94].4   // IO-Link Port 5 - Device ID (INT bit4)
           TBEN_L4_8IOL:C.Data[94].5   // IO-Link Port 5 - Device ID (INT bit5)
           TBEN_L4_8IOL:C.Data[94].6   // IO-Link Port 5 - Device ID (INT bit6)
           TBEN_L4_8IOL:C.Data[94].7   // IO-Link Port 5 - Device ID (INT bit7)
           TBEN_L4_8IOL:C.Data[95]   // IO-Link Port 5 - Device ID
           TBEN_L4_8IOL:C.Data[95].0   // IO-Link Port 5 - Device ID (INT bit8)
           TBEN_L4_8IOL:C.Data[95].1   // IO-Link Port 5 - Device ID (INT bit9)
           TBEN_L4_8IOL:C.Data[95].2   // IO-Link Port 5 - Device ID (INT bit10)
           TBEN_L4_8IOL:C.Data[95].3   // IO-Link Port 5 - Device ID (INT bit11)
           TBEN_L4_8IOL:C.Data[95].4   // IO-Link Port 5 - Device ID (INT bit12)
           TBEN_L4_8IOL:C.Data[95].5   // IO-Link Port 5 - Device ID (INT bit13)
           TBEN_L4_8IOL:C.Data[95].6   // IO-Link Port 5 - Device ID (INT bit14)
           TBEN_L4_8IOL:C.Data[95].7   // IO-Link Port 5 - Device ID (INT bit15)
           TBEN_L4_8IOL:C.Data[96]   // IO-Link Port 5 - Device ID
           TBEN_L4_8IOL:C.Data[96].0   // IO-Link Port 5 - Device ID (INT bit16)
           TBEN_L4_8IOL:C.Data[96].1   // IO-Link Port 5 - Device ID (INT bit17)
           TBEN_L4_8IOL:C.Data[96].2   // IO-Link Port 5 - Device ID (INT bit18)
           TBEN_L4_8IOL:C.Data[96].3   // IO-Link Port 5 - Device ID (INT bit19)
           TBEN_L4_8IOL:C.Data[96].4   // IO-Link Port 5 - Device ID (INT bit20)
           TBEN_L4_8IOL:C.Data[96].5   // IO-Link Port 5 - Device ID (INT bit21)
           TBEN_L4_8IOL:C.Data[96].6   // IO-Link Port 5 - Device ID (INT bit22)
           TBEN_L4_8IOL:C.Data[96].7   // IO-Link Port 5 - Device ID (INT bit23)
           TBEN_L4_8IOL:C.Data[97]   // IO-Link Port 5 - Device ID
           TBEN_L4_8IOL:C.Data[97].0   // IO-Link Port 5 - Device ID (INT bit24)
           TBEN_L4_8IOL:C.Data[97].1   // IO-Link Port 5 - Device ID (INT bit25)
           TBEN_L4_8IOL:C.Data[97].2   // IO-Link Port 5 - Device ID (INT bit26)
           TBEN_L4_8IOL:C.Data[97].3   // IO-Link Port 5 - Device ID (INT bit27)
           TBEN_L4_8IOL:C.Data[97].4   // IO-Link Port 5 - Device ID (INT bit28)
           TBEN_L4_8IOL:C.Data[97].5   // IO-Link Port 5 - Device ID (INT bit29)
           TBEN_L4_8IOL:C.Data[97].6   // IO-Link Port 5 - Device ID (INT bit30)
           TBEN_L4_8IOL:C.Data[97].7   // IO-Link Port 5 - Device ID (INT bit31)
           TBEN_L4_8IOL:C.Data[98]   // IO-Link Port 6 - Operation mode
           TBEN_L4_8IOL:C.Data[98].0   // IO-Link Port 6 - Operation mode (ENUM bit0): 0000=IO-Link without validation, 0001=IO-Link with family compatible device
           TBEN_L4_8IOL:C.Data[98].1   // IO-Link Port 6 - Operation mode (ENUM bit1): 0010=IO-Link with compatible device, 0011=IO-Link with identical device
           TBEN_L4_8IOL:C.Data[98].2   // IO-Link Port 6 - Operation mode (ENUM bit2): 0100=DI (with parameter access)
           TBEN_L4_8IOL:C.Data[98].3   // IO-Link Port 6 - Operation mode (ENUM bit3): 1000=DI
           TBEN_L4_8IOL:C.Data[98].4   // Reserved
           TBEN_L4_8IOL:C.Data[98].5   // Reserved
           TBEN_L4_8IOL:C.Data[98].6   // Reserved
           TBEN_L4_8IOL:C.Data[98].7   // Reserved
           TBEN_L4_8IOL:C.Data[99]   // IO-Link Port 6 - Data storage mode
           TBEN_L4_8IOL:C.Data[99].0   // IO-Link Port 6 - Data storage mode (ENUM bit0): 00=activated, 01=overwrite
           TBEN_L4_8IOL:C.Data[99].1   // IO-Link Port 6 - Data storage mode (ENUM bit1): 10=read in, 11=deactivated, clear
           TBEN_L4_8IOL:C.Data[99].2   // Reserved
           TBEN_L4_8IOL:C.Data[99].3   // Reserved
           TBEN_L4_8IOL:C.Data[99].4   // Reserved
           TBEN_L4_8IOL:C.Data[99].5   // Reserved
           TBEN_L4_8IOL:C.Data[99].6   // Reserved
           TBEN_L4_8IOL:C.Data[99].7   // Reserved
           TBEN_L4_8IOL:C.Data[9]   // Quick Connect, Eth Custom Setup, LED-behavior (PWR) at V2 undervoltage
           TBEN_L4_8IOL:C.Data[9].0   // Quick Connect: 0=disable, 1=enable
           TBEN_L4_8IOL:C.Data[9].1   // Eth 1 Custom Setup: 0=Auto-negotiate, 1=100BT/FD
           TBEN_L4_8IOL:C.Data[9].2   // Eth 2 Custom Setup: 0=Auto-negotiate, 1=100BT/FD
           TBEN_L4_8IOL:C.Data[9].3   // LED-behavior (PWR) at V2 undervoltage: 0=Red, 1=Green
           TBEN_L4_8IOL:C.Data[9].4   // Reserved
           TBEN_L4_8IOL:C.Data[9].5   // Reserved
           TBEN_L4_8IOL:C.Data[9].6   // Reserved
           TBEN_L4_8IOL:C.Data[9].7   // Reserved
END_MODULES
